DECL LDAT LCPDAT2987={VEL 2.00000,ACC 100.000,APO_DIST 500.000,APO_FAC 50.0000,AXIS_VEL 100.000,AXIS_ACC 100.000,ORI_TYP #VAR,CIRC_TYP #BASE,JERK_FAC 50.0000,GEAR_JERK 100.000,EXAX_IGN 0}
DECL E6POS XP2988={X 377.0,Y 306.0,Z -17.64,A -180,B 0,C 180,S 2,T 10,E1 0.0,E2 0.0,E3 0.0,E4 0.0,E5 0.0,E6 0.0}
DECL FDAT FP2988={TOOL_NO 1,BASE_NO 0,IPO_FRAME #BASE,POINT2[] " "}
DECL LDAT LCPDAT2988={VEL 2.00000,ACC 100.000,APO_DIST 500.000,APO_FAC 50.0000,AXIS_VEL 100.000,AXIS_ACC 100.000,ORI_TYP #VAR,CIRC_TYP #BASE,JERK_FAC 50.0000,GEAR_JERK 100.000,EXAX_IGN 0}
DECL E6POS XP2989={X 377.0,Y 306.0,Z -17.64,A -180,B 0,C 180,S 2,T 10,E1 0.0,E2 0.0,E3 0.0,E4 0.0,E5 0.0,E6 0.0}
DECL FDAT FP2989={TOOL_NO 1,BASE_NO 0,IPO_FRAME #BASE,POINT2[] " "}
DECL LDAT LCPDAT2989={VEL 2.00000,ACC 100.000,APO_DIST 500.000,APO_FAC 50.0000,AXIS_VEL 100.000,AXIS_ACC 100.000,ORI_TYP #VAR,CIRC_TYP #BASE,JERK_FAC 50.0000,GEAR_JERK 100.000,EXAX_IGN 0}
DECL E6POS XP2990={X 379.0,Y 306.0,Z -17.64,A -180,B 0,C 180,S 2,T 10,E1 0.0,E2 0.0,E3 0.0,E4 0.0,E5 0.0,E6 0.0}
DECL FDAT FP2990={TOOL_NO 1,BASE_NO 0,IPO_FRAME #BASE,POINT2[] " "}
DECL LDAT LCPDAT2990={VEL 2.00000,ACC 100.000,APO_DIST 500.000,APO_FAC 50.0000,AXIS_VEL 100.000,AXIS_ACC 100.000,ORI_TYP #VAR,CIRC_TYP #BASE,JERK_FAC 50.0000,GEAR_JERK 100.000,EXAX_IGN 0}
DECL E6POS XP2991={X 379.0,Y 306.0,Z -17.64,A -180,B 0,C 180,S 2,T 10,E1 0.0,E2 0.0,E3 0.0,E4 0.0,E5 0.0,E6 0.0}
DECL FDAT FP2991={TOOL_NO 1,BASE_NO 0,IPO_FRAME #BASE,POINT2[] " "}
DECL LDAT LCPDAT2991={VEL 2.00000,ACC 100.000,APO_DIST 500.000,APO_FAC 50.0000,AXIS_VEL 100.000,AXIS_ACC 100.000,ORI_TYP #VAR,CIRC_TYP #BASE,JERK_FAC 50.0000,GEAR_JERK 100.000,EXAX_IGN 0}
DECL E6POS XP2992={X 380.0,Y 304.0,Z -17.64,A -180,B 0,C 180,S 2,T 10,E1 0.0,E2 0.0,E3 0.0,E4 0.0,E5 0.0,E6 0.0}
DECL FDAT FP2992={TOOL_NO 1,BASE_NO 0,IPO_FRAME #BASE,POINT2[] " "}
DECL LDAT LCPDAT2992={VEL 2.00000,ACC 100.000,APO_DIST 500.000,APO_FAC 50.0000,AXIS_VEL 100.000,AXIS_ACC 100.000,ORI_TYP #VAR,CIRC_TYP #BASE,JERK_FAC 50.0000,GEAR_JERK 100.000,EXAX_IGN 0}
DECL E6POS XP2993={X 380.0,Y 304.0,Z -17.64,A -180,B 0,C 180,S 2,T 10,E1 0.0,E2 0.0,E3 0.0,E4 0.0,E5 0.0,E6 0.0}
DECL FDAT FP2993={TOOL_NO 1,BASE_NO 0,IPO_FRAME #BASE,POINT2[] " "}
DECL LDAT LCPDAT2993={VEL 2.00000,ACC 100.000,APO_DIST 500.000,APO_FAC 50.0000,AXIS_VEL 100.000,AXIS_ACC 100.000,ORI_TYP #VAR,CIRC_TYP #BASE,JERK_FAC 50.0000,GEAR_JERK 100.000,EXAX_IGN 0}
DECL E6POS XP2994={X 381.0,Y 313.0,Z -17.64,A -180,B 0,C 180,S 2,T 10,E1 0.0,E2 0.0,E3 0.0,E4 0.0,E5 0.0,E6 0.0}
DECL FDAT FP2994={TOOL_NO 1,BASE_NO 0,IPO_FRAME #BASE,POINT2[] " "}
DECL LDAT LCPDAT2994={VEL 2.00000,ACC 100.000,APO_DIST 500.000,APO_FAC 50.0000,AXIS_VEL 100.000,AXIS_ACC 100.000,ORI_TYP #VAR,CIRC_TYP #BASE,JERK_FAC 50.0000,GEAR_JERK 100.000,EXAX_IGN 0}
DECL E6POS XP2995={X 381.0,Y 313.0,Z -17.64,A -180,B 0,C 180,S 2,T 10,E1 0.0,E2 0.0,E3 0.0,E4 0.0,E5 0.0,E6 0.0}
DECL FDAT FP2995={TOOL_NO 1,BASE_NO 0,IPO_FRAME #BASE,POINT2[] " "}
DECL LDAT LCPDAT2995={VEL 2.00000,ACC 100.000,APO_DIST 500.000,APO_FAC 50.0000,AXIS_VEL 100.000,AXIS_ACC 100.000,ORI_TYP #VAR,CIRC_TYP #BASE,JERK_FAC 50.0000,GEAR_JERK 100.000,EXAX_IGN 0}
DECL E6POS XP2996={X 379.0,Y 315.0,Z -17.64,A -180,B 0,C 180,S 2,T 10,E1 0.0,E2 0.0,E3 0.0,E4 0.0,E5 0.0,E6 0.0}
DECL FDAT FP2996={TOOL_NO 1,BASE_NO 0,IPO_FRAME #BASE,POINT2[] " "}
DECL LDAT LCPDAT2996={VEL 2.00000,ACC 100.000,APO_DIST 500.000,APO_FAC 50.0000,AXIS_VEL 100.000,AXIS_ACC 100.000,ORI_TYP #VAR,CIRC_TYP #BASE,JERK_FAC 50.0000,GEAR_JERK 100.000,EXAX_IGN 0}
DECL E6POS XP2997={X 379.0,Y 315.0,Z -17.64,A -180,B 0,C 180,S 2,T 10,E1 0.0,E2 0.0,E3 0.0,E4 0.0,E5 0.0,E6 0.0}
DECL FDAT FP2997={TOOL_NO 1,BASE_NO 0,IPO_FRAME #BASE,POINT2[] " "}
DECL LDAT LCPDAT2997={VEL 2.00000,ACC 100.000,APO_DIST 500.000,APO_FAC 50.0000,AXIS_VEL 100.000,AXIS_ACC 100.000,ORI_TYP #VAR,CIRC_TYP #BASE,JERK_FAC 50.0000,GEAR_JERK 100.000,EXAX_IGN 0}
DECL E6POS XP2998={X 375.0,Y 315.0,Z -17.64,A -180,B 0,C 180,S 2,T 10,E1 0.0,E2 0.0,E3 0.0,E4 0.0,E5 0.0,E6 0.0}
DECL FDAT FP2998={TOOL_NO 1,BASE_NO 0,IPO_FRAME #BASE,POINT2[] " "}
DECL LDAT LCPDAT2998={VEL 2.00000,ACC 100.000,APO_DIST 500.000,APO_FAC 50.0000,AXIS_VEL 100.000,AXIS_ACC 100.000,ORI_TYP #VAR,CIRC_TYP #BASE,JERK_FAC 50.0000,GEAR_JERK 100.000,EXAX_IGN 0}
DECL E6POS XP2999={X 375.0,Y 315.0,Z -17.64,A -180,B 0,C 180,S 2,T 10,E1 0.0,E2 0.0,E3 0.0,E4 0.0,E5 0.0,E6 0.0}
DECL FDAT FP2999={TOOL_NO 1,BASE_NO 0,IPO_FRAME #BASE,POINT2[] " "}
DECL LDAT LCPDAT2999={VEL 2.00000,ACC 100.000,APO_DIST 500.000,APO_FAC 50.0000,AXIS_VEL 100.000,AXIS_ACC 100.000,ORI_TYP #VAR,CIRC_TYP #BASE,JERK_FAC 50.0000,GEAR_JERK 100.000,EXAX_IGN 0}
DECL E6POS XP3000={X 375.0,Y 317.0,Z -17.64,A -180,B 0,C 180,S 2,T 10,E1 0.0,E2 0.0,E3 0.0,E4 0.0,E5 0.0,E6 0.0}
DECL FDAT FP3000={TOOL_NO 1,BASE_NO 0,IPO_FRAME #BASE,POINT2[] " "}
DECL LDAT LCPDAT3000={VEL 2.00000,ACC 100.000,APO_DIST 500.000,APO_FAC 50.0000,AXIS_VEL 100.000,AXIS_ACC 100.000,ORI_TYP #VAR,CIRC_TYP #BASE,JERK_FAC 50.0000,GEAR_JERK 100.000,EXAX_IGN 0}
DECL E6POS XP3001={X 375.0,Y 317.0,Z -17.64,A -180,B 0,C 180,S 2,T 10,E1 0.0,E2 0.0,E3 0.0,E4 0.0,E5 0.0,E6 0.0}
DECL FDAT FP3001={TOOL_NO 1,BASE_NO 0,IPO_FRAME #BASE,POINT2[] " "}
DECL LDAT LCPDAT3001={VEL 2.00000,ACC 100.000,APO_DIST 500.000,APO_FAC 50.0000,AXIS_VEL 100.000,AXIS_ACC 100.000,ORI_TYP #VAR,CIRC_TYP #BASE,JERK_FAC 50.0000,GEAR_JERK 100.000,EXAX_IGN 0}
DECL E6POS XP3002={X 376.0,Y 320.0,Z -17.64,A -180,B 0,C 180,S 2,T 10,E1 0.0,E2 0.0,E3 0.0,E4 0.0,E5 0.0,E6 0.0}
DECL FDAT FP3002={TOOL_NO 1,BASE_NO 0,IPO_FRAME #BASE,POINT2[] " "}
DECL LDAT LCPDAT3002={VEL 2.00000,ACC 100.000,APO_DIST 500.000,APO_FAC 50.0000,AXIS_VEL 100.000,AXIS_ACC 100.000,ORI_TYP #VAR,CIRC_TYP #BASE,JERK_FAC 50.0000,GEAR_JERK 100.000,EXAX_IGN 0}
DECL E6POS XP3003={X 376.0,Y 320.0,Z -17.64,A -180,B 0,C 180,S 2,T 10,E1 0.0,E2 0.0,E3 0.0,E4 0.0,E5 0.0,E6 0.0}
DECL FDAT FP3003={TOOL_NO 1,BASE_NO 0,IPO_FRAME #BASE,POINT2[] " "}
DECL LDAT LCPDAT3003={VEL 2.00000,ACC 100.000,APO_DIST 500.000,APO_FAC 50.0000,AXIS_VEL 100.000,AXIS_ACC 100.000,ORI_TYP #VAR,CIRC_TYP #BASE,JERK_FAC 50.0000,GEAR_JERK 100.000,EXAX_IGN 0}
DECL E6POS XP3004={X 378.0,Y 322.0,Z -17.64,A -180,B 0,C 180,S 2,T 10,E1 0.0,E2 0.0,E3 0.0,E4 0.0,E5 0.0,E6 0.0}
DECL FDAT FP3004={TOOL_NO 1,BASE_NO 0,IPO_FRAME #BASE,POINT2[] " "}
DECL LDAT LCPDAT3004={VEL 2.00000,ACC 100.000,APO_DIST 500.000,APO_FAC 50.0000,AXIS_VEL 100.000,AXIS_ACC 100.000,ORI_TYP #VAR,CIRC_TYP #BASE,JERK_FAC 50.0000,GEAR_JERK 100.000,EXAX_IGN 0}
DECL E6POS XP3005={X 378.0,Y 322.0,Z -17.64,A -180,B 0,C 180,S 2,T 10,E1 0.0,E2 0.0,E3 0.0,E4 0.0,E5 0.0,E6 0.0}
DECL FDAT FP3005={TOOL_NO 1,BASE_NO 0,IPO_FRAME #BASE,POINT2[] " "}
DECL LDAT LCPDAT3005={VEL 2.00000,ACC 100.000,APO_DIST 500.000,APO_FAC 50.0000,AXIS_VEL 100.000,AXIS_ACC 100.000,ORI_TYP #VAR,CIRC_TYP #BASE,JERK_FAC 50.0000,GEAR_JERK 100.000,EXAX_IGN 0}
DECL E6POS XP3006={X 379.0,Y 326.0,Z -17.64,A -180,B 0,C 180,S 2,T 10,E1 0.0,E2 0.0,E3 0.0,E4 0.0,E5 0.0,E6 0.0}
DECL FDAT FP3006={TOOL_NO 1,BASE_NO 0,IPO_FRAME #BASE,POINT2[] " "}
DECL LDAT LCPDAT3006={VEL 2.00000,ACC 100.000,APO_DIST 500.000,APO_FAC 50.0000,AXIS_VEL 100.000,AXIS_ACC 100.000,ORI_TYP #VAR,CIRC_TYP #BASE,JERK_FAC 50.0000,GEAR_JERK 100.000,EXAX_IGN 0}
DECL E6POS XP3007={X 379.0,Y 326.0,Z -17.64,A -180,B 0,C 180,S 2,T 10,E1 0.0,E2 0.0,E3 0.0,E4 0.0,E5 0.0,E6 0.0}
DECL FDAT FP3007={TOOL_NO 1,BASE_NO 0,IPO_FRAME #BASE,POINT2[] " "}
DECL LDAT LCPDAT3007={VEL 2.00000,ACC 100.000,APO_DIST 500.000,APO_FAC 50.0000,AXIS_VEL 100.000,AXIS_ACC 100.000,ORI_TYP #VAR,CIRC_TYP #BASE,JERK_FAC 50.0000,GEAR_JERK 100.000,EXAX_IGN 0}
DECL E6POS XP3008={X 378.0,Y 330.0,Z -17.64,A -180,B 0,C 180,S 2,T 10,E1 0.0,E2 0.0,E3 0.0,E4 0.0,E5 0.0,E6 0.0}
DECL FDAT FP3008={TOOL_NO 1,BASE_NO 0,IPO_FRAME #BASE,POINT2[] " "}
DECL LDAT LCPDAT3008={VEL 2.00000,ACC 100.000,APO_DIST 500.000,APO_FAC 50.0000,AXIS_VEL 100.000,AXIS_ACC 100.000,ORI_TYP #VAR,CIRC_TYP #BASE,JERK_FAC 50.0000,GEAR_JERK 100.000,EXAX_IGN 0}
DECL E6POS XP3009={X 378.0,Y 330.0,Z -17.64,A -180,B 0,C 180,S 2,T 10,E1 0.0,E2 0.0,E3 0.0,E4 0.0,E5 0.0,E6 0.0}
DECL FDAT FP3009={TOOL_NO 1,BASE_NO 0,IPO_FRAME #BASE,POINT2[] " "}
DECL LDAT LCPDAT3009={VEL 2.00000,ACC 100.000,APO_DIST 500.000,APO_FAC 50.0000,AXIS_VEL 100.000,AXIS_ACC 100.000,ORI_TYP #VAR,CIRC_TYP #BASE,JERK_FAC 50.0000,GEAR_JERK 100.000,EXAX_IGN 0}
DECL E6POS XP3010={X 376.0,Y 329.0,Z -17.64,A -180,B 0,C 180,S 2,T 10,E1 0.0,E2 0.0,E3 0.0,E4 0.0,E5 0.0,E6 0.0}
DECL FDAT FP3010={TOOL_NO 1,BASE_NO 0,IPO_FRAME #BASE,POINT2[] " "}
DECL LDAT LCPDAT3010={VEL 2.00000,ACC 100.000,APO_DIST 500.000,APO_FAC 50.0000,AXIS_VEL 100.000,AXIS_ACC 100.000,ORI_TYP #VAR,CIRC_TYP #BASE,JERK_FAC 50.0000,GEAR_JERK 100.000,EXAX_IGN 0}
DECL E6POS XP3011={X 376.0,Y 329.0,Z -17.64,A -180,B 0,C 180,S 2,T 10,E1 0.0,E2 0.0,E3 0.0,E4 0.0,E5 0.0,E6 0.0}
DECL FDAT FP3011={TOOL_NO 1,BASE_NO 0,IPO_FRAME #BASE,POINT2[] " "}
DECL LDAT LCPDAT3011={VEL 2.00000,ACC 100.000,APO_DIST 500.000,APO_FAC 50.0000,AXIS_VEL 100.000,AXIS_ACC 100.000,ORI_TYP #VAR,CIRC_TYP #BASE,JERK_FAC 50.0000,GEAR_JERK 100.000,EXAX_IGN 0}
DECL E6POS XP3012={X 376.0,Y 334.0,Z -17.64,A -180,B 0,C 180,S 2,T 10,E1 0.0,E2 0.0,E3 0.0,E4 0.0,E5 0.0,E6 0.0}
DECL FDAT FP3012={TOOL_NO 1,BASE_NO 0,IPO_FRAME #BASE,POINT2[] " "}
DECL LDAT LCPDAT3012={VEL 2.00000,ACC 100.000,APO_DIST 500.000,APO_FAC 50.0000,AXIS_VEL 100.000,AXIS_ACC 100.000,ORI_TYP #VAR,CIRC_TYP #BASE,JERK_FAC 50.0000,GEAR_JERK 100.000,EXAX_IGN 0}
DECL E6POS XP3013={X 376.0,Y 334.0,Z -17.64,A -180,B 0,C 180,S 2,T 10,E1 0.0,E2 0.0,E3 0.0,E4 0.0,E5 0.0,E6 0.0}
DECL FDAT FP3013={TOOL_NO 1,BASE_NO 0,IPO_FRAME #BASE,POINT2[] " "}
DECL LDAT LCPDAT3013={VEL 2.00000,ACC 100.000,APO_DIST 500.000,APO_FAC 50.0000,AXIS_VEL 100.000,AXIS_ACC 100.000,ORI_TYP #VAR,CIRC_TYP #BASE,JERK_FAC 50.0000,GEAR_JERK 100.000,EXAX_IGN 0}
DECL E6POS XP3014={X 378.0,Y 333.0,Z -17.64,A -180,B 0,C 180,S 2,T 10,E1 0.0,E2 0.0,E3 0.0,E4 0.0,E5 0.0,E6 0.0}
DECL FDAT FP3014={TOOL_NO 1,BASE_NO 0,IPO_FRAME #BASE,POINT2[] " "}
DECL LDAT LCPDAT3014={VEL 2.00000,ACC 100.000,APO_DIST 500.000,APO_FAC 50.0000,AXIS_VEL 100.000,AXIS_ACC 100.000,ORI_TYP #VAR,CIRC_TYP #BASE,JERK_FAC 50.0000,GEAR_JERK 100.000,EXAX_IGN 0}
DECL E6POS XP3015={X 378.0,Y 333.0,Z -17.64,A -180,B 0,C 180,S 2,T 10,E1 0.0,E2 0.0,E3 0.0,E4 0.0,E5 0.0,E6 0.0}
DECL FDAT FP3015={TOOL_NO 1,BASE_NO 0,IPO_FRAME #BASE,POINT2[] " "}
DECL LDAT LCPDAT3015={VEL 2.00000,ACC 100.000,APO_DIST 500.000,APO_FAC 50.0000,AXIS_VEL 100.000,AXIS_ACC 100.000,ORI_TYP #VAR,CIRC_TYP #BASE,JERK_FAC 50.0000,GEAR_JERK 100.000,EXAX_IGN 0}
DECL E6POS XP3016={X 378.0,Y 337.0,Z -17.64,A -180,B 0,C 180,S 2,T 10,E1 0.0,E2 0.0,E3 0.0,E4 0.0,E5 0.0,E6 0.0}
DECL FDAT FP3016={TOOL_NO 1,BASE_NO 0,IPO_FRAME #BASE,POINT2[] " "}
DECL LDAT LCPDAT3016={VEL 2.00000,ACC 100.000,APO_DIST 500.000,APO_FAC 50.0000,AXIS_VEL 100.000,AXIS_ACC 100.000,ORI_TYP #VAR,CIRC_TYP #BASE,JERK_FAC 50.0000,GEAR_JERK 100.000,EXAX_IGN 0}
DECL E6POS XP3017={X 378.0,Y 337.0,Z -17.64,A -180,B 0,C 180,S 2,T 10,E1 0.0,E2 0.0,E3 0.0,E4 0.0,E5 0.0,E6 0.0}
DECL FDAT FP3017={TOOL_NO 1,BASE_NO 0,IPO_FRAME #BASE,POINT2[] " "}
DECL LDAT LCPDAT3017={VEL 2.00000,ACC 100.000,APO_DIST 500.000,APO_FAC 50.0000,AXIS_VEL 100.000,AXIS_ACC 100.000,ORI_TYP #VAR,CIRC_TYP #BASE,JERK_FAC 50.0000,GEAR_JERK 100.000,EXAX_IGN 0}
DECL E6POS XP3018={X 377.0,Y 336.0,Z -17.64,A -180,B 0,C 180,S 2,T 10,E1 0.0,E2 0.0,E3 0.0,E4 0.0,E5 0.0,E6 0.0}
DECL FDAT FP3018={TOOL_NO 1,BASE_NO 0,IPO_FRAME #BASE,POINT2[] " "}
DECL LDAT LCPDAT3018={VEL 2.00000,ACC 100.000,APO_DIST 500.000,APO_FAC 50.0000,AXIS_VEL 100.000,AXIS_ACC 100.000,ORI_TYP #VAR,CIRC_TYP #BASE,JERK_FAC 50.0000,GEAR_JERK 100.000,EXAX_IGN 0}
DECL E6POS XP3019={X 377.0,Y 336.0,Z -17.64,A -180,B 0,C 180,S 2,T 10,E1 0.0,E2 0.0,E3 0.0,E4 0.0,E5 0.0,E6 0.0}
DECL FDAT FP3019={TOOL_NO 1,BASE_NO 0,IPO_FRAME #BASE,POINT2[] " "}
DECL LDAT LCPDAT3019={VEL 2.00000,ACC 100.000,APO_DIST 500.000,APO_FAC 50.0000,AXIS_VEL 100.000,AXIS_ACC 100.000,ORI_TYP #VAR,CIRC_TYP #BASE,JERK_FAC 50.0000,GEAR_JERK 100.000,EXAX_IGN 0}
DECL E6POS XP3020={X 376.0,Y 339.0,Z -17.64,A -180,B 0,C 180,S 2,T 10,E1 0.0,E2 0.0,E3 0.0,E4 0.0,E5 0.0,E6 0.0}
DECL FDAT FP3020={TOOL_NO 1,BASE_NO 0,IPO_FRAME #BASE,POINT2[] " "}
DECL LDAT LCPDAT3020={VEL 2.00000,ACC 100.000,APO_DIST 500.000,APO_FAC 50.0000,AXIS_VEL 100.000,AXIS_ACC 100.000,ORI_TYP #VAR,CIRC_TYP #BASE,JERK_FAC 50.0000,GEAR_JERK 100.000,EXAX_IGN 0}
DECL E6POS XP3021={X 376.0,Y 339.0,Z -17.64,A -180,B 0,C 180,S 2,T 10,E1 0.0,E2 0.0,E3 0.0,E4 0.0,E5 0.0,E6 0.0}
DECL FDAT FP3021={TOOL_NO 1,BASE_NO 0,IPO_FRAME #BASE,POINT2[] " "}
DECL LDAT LCPDAT3021={VEL 2.00000,ACC 100.000,APO_DIST 500.000,APO_FAC 50.0000,AXIS_VEL 100.000,AXIS_ACC 100.000,ORI_TYP #VAR,CIRC_TYP #BASE,JERK_FAC 50.0000,GEAR_JERK 100.000,EXAX_IGN 0}
DECL E6POS XP3022={X 374.0,Y 341.0,Z -17.64,A -180,B 0,C 180,S 2,T 10,E1 0.0,E2 0.0,E3 0.0,E4 0.0,E5 0.0,E6 0.0}
DECL FDAT FP3022={TOOL_NO 1,BASE_NO 0,IPO_FRAME #BASE,POINT2[] " "}
DECL LDAT LCPDAT3022={VEL 2.00000,ACC 100.000,APO_DIST 500.000,APO_FAC 50.0000,AXIS_VEL 100.000,AXIS_ACC 100.000,ORI_TYP #VAR,CIRC_TYP #BASE,JERK_FAC 50.0000,GEAR_JERK 100.000,EXAX_IGN 0}
DECL E6POS XP3023={X 374.0,Y 341.0,Z -17.64,A -180,B 0,C 180,S 2,T 10,E1 0.0,E2 0.0,E3 0.0,E4 0.0,E5 0.0,E6 0.0}
DECL FDAT FP3023={TOOL_NO 1,BASE_NO 0,IPO_FRAME #BASE,POINT2[] " "}
DECL LDAT LCPDAT3023={VEL 2.00000,ACC 100.000,APO_DIST 500.000,APO_FAC 50.0000,AXIS_VEL 100.000,AXIS_ACC 100.000,ORI_TYP #VAR,CIRC_TYP #BASE,JERK_FAC 50.0000,GEAR_JERK 100.000,EXAX_IGN 0}
DECL E6POS XP3024={X 372.0,Y 338.0,Z -17.64,A -180,B 0,C 180,S 2,T 10,E1 0.0,E2 0.0,E3 0.0,E4 0.0,E5 0.0,E6 0.0}
DECL FDAT FP3024={TOOL_NO 1,BASE_NO 0,IPO_FRAME #BASE,POINT2[] " "}
DECL LDAT LCPDAT3024={VEL 2.00000,ACC 100.000,APO_DIST 500.000,APO_FAC 50.0000,AXIS_VEL 100.000,AXIS_ACC 100.000,ORI_TYP #VAR,CIRC_TYP #BASE,JERK_FAC 50.0000,GEAR_JERK 100.000,EXAX_IGN 0}
DECL E6POS XP3025={X 372.0,Y 338.0,Z -17.64,A -180,B 0,C 180,S 2,T 10,E1 0.0,E2 0.0,E3 0.0,E4 0.0,E5 0.0,E6 0.0}
DECL FDAT FP3025={TOOL_NO 1,BASE_NO 0,IPO_FRAME #BASE,POINT2[] " "}
DECL LDAT LCPDAT3025={VEL 2.00000,ACC 100.000,APO_DIST 500.000,APO_FAC 50.0000,AXIS_VEL 100.000,AXIS_ACC 100.000,ORI_TYP #VAR,CIRC_TYP #BASE,JERK_FAC 50.0000,GEAR_JERK 100.000,EXAX_IGN 0}
DECL E6POS XP3026={X 374.0,Y 337.0,Z -17.64,A -180,B 0,C 180,S 2,T 10,E1 0.0,E2 0.0,E3 0.0,E4 0.0,E5 0.0,E6 0.0}
DECL FDAT FP3026={TOOL_NO 1,BASE_NO 0,IPO_FRAME #BASE,POINT2[] " "}
DECL LDAT LCPDAT3026={VEL 2.00000,ACC 100.000,APO_DIST 500.000,APO_FAC 50.0000,AXIS_VEL 100.000,AXIS_ACC 100.000,ORI_TYP #VAR,CIRC_TYP #BASE,JERK_FAC 50.0000,GEAR_JERK 100.000,EXAX_IGN 0}
DECL E6POS XP3027={X 374.0,Y 337.0,Z -17.64,A -180,B 0,C 180,S 2,T 10,E1 0.0,E2 0.0,E3 0.0,E4 0.0,E5 0.0,E6 0.0}
DECL FDAT FP3027={TOOL_NO 1,BASE_NO 0,IPO_FRAME #BASE,POINT2[] " "}
DECL LDAT LCPDAT3027={VEL 2.00000,ACC 100.000,APO_DIST 500.000,APO_FAC 50.0000,AXIS_VEL 100.000,AXIS_ACC 100.000,ORI_TYP #VAR,CIRC_TYP #BASE,JERK_FAC 50.0000,GEAR_JERK 100.000,EXAX_IGN 0}
DECL E6POS XP3028={X 372.0,Y 338.0,Z -17.64,A -180,B 0,C 180,S 2,T 10,E1 0.0,E2 0.0,E3 0.0,E4 0.0,E5 0.0,E6 0.0}
DECL FDAT FP3028={TOOL_NO 1,BASE_NO 0,IPO_FRAME #BASE,POINT2[] " "}
DECL LDAT LCPDAT3028={VEL 2.00000,ACC 100.000,APO_DIST 500.000,APO_FAC 50.0000,AXIS_VEL 100.000,AXIS_ACC 100.000,ORI_TYP #VAR,CIRC_TYP #BASE,JERK_FAC 50.0000,GEAR_JERK 100.000,EXAX_IGN 0}
DECL E6POS XP3029={X 372.0,Y 338.0,Z -17.64,A -180,B 0,C 180,S 2,T 10,E1 0.0,E2 0.0,E3 0.0,E4 0.0,E5 0.0,E6 0.0}
DECL FDAT FP3029={TOOL_NO 1,BASE_NO 0,IPO_FRAME #BASE,POINT2[] " "}
DECL LDAT LCPDAT3029={VEL 2.00000,ACC 100.000,APO_DIST 500.000,APO_FAC 50.0000,AXIS_VEL 100.000,AXIS_ACC 100.000,ORI_TYP #VAR,CIRC_TYP #BASE,JERK_FAC 50.0000,GEAR_JERK 100.000,EXAX_IGN 0}
DECL E6POS XP3030={X 373.0,Y 341.0,Z -17.64,A -180,B 0,C 180,S 2,T 10,E1 0.0,E2 0.0,E3 0.0,E4 0.0,E5 0.0,E6 0.0}
DECL FDAT FP3030={TOOL_NO 1,BASE_NO 0,IPO_FRAME #BASE,POINT2[] " "}
DECL LDAT LCPDAT3030={VEL 2.00000,ACC 100.000,APO_DIST 500.000,APO_FAC 50.0000,AXIS_VEL 100.000,AXIS_ACC 100.000,ORI_TYP #VAR,CIRC_TYP #BASE,JERK_FAC 50.0000,GEAR_JERK 100.000,EXAX_IGN 0}
DECL E6POS XP3031={X 373.0,Y 341.0,Z -17.64,A -180,B 0,C 180,S 2,T 10,E1 0.0,E2 0.0,E3 0.0,E4 0.0,E5 0.0,E6 0.0}
DECL FDAT FP3031={TOOL_NO 1,BASE_NO 0,IPO_FRAME #BASE,POINT2[] " "}
DECL LDAT LCPDAT3031={VEL 2.00000,ACC 100.000,APO_DIST 500.000,APO_FAC 50.0000,AXIS_VEL 100.000,AXIS_ACC 100.000,ORI_TYP #VAR,CIRC_TYP #BASE,JERK_FAC 50.0000,GEAR_JERK 100.000,EXAX_IGN 0}
DECL E6POS XP3032={X 375.0,Y 342.0,Z -17.64,A -180,B 0,C 180,S 2,T 10,E1 0.0,E2 0.0,E3 0.0,E4 0.0,E5 0.0,E6 0.0}
DECL FDAT FP3032={TOOL_NO 1,BASE_NO 0,IPO_FRAME #BASE,POINT2[] " "}
DECL LDAT LCPDAT3032={VEL 2.00000,ACC 100.000,APO_DIST 500.000,APO_FAC 50.0000,AXIS_VEL 100.000,AXIS_ACC 100.000,ORI_TYP #VAR,CIRC_TYP #BASE,JERK_FAC 50.0000,GEAR_JERK 100.000,EXAX_IGN 0}
DECL E6POS XP3033={X 375.0,Y 342.0,Z -17.64,A -180,B 0,C 180,S 2,T 10,E1 0.0,E2 0.0,E3 0.0,E4 0.0,E5 0.0,E6 0.0}
DECL FDAT FP3033={TOOL_NO 1,BASE_NO 0,IPO_FRAME #BASE,POINT2[] " "}
DECL LDAT LCPDAT3033={VEL 2.00000,ACC 100.000,APO_DIST 500.000,APO_FAC 50.0000,AXIS_VEL 100.000,AXIS_ACC 100.000,ORI_TYP #VAR,CIRC_TYP #BASE,JERK_FAC 50.0000,GEAR_JERK 100.000,EXAX_IGN 0}
DECL E6POS XP3034={X 375.0,Y 344.0,Z -17.64,A -180,B 0,C 180,S 2,T 10,E1 0.0,E2 0.0,E3 0.0,E4 0.0,E5 0.0,E6 0.0}
DECL FDAT FP3034={TOOL_NO 1,BASE_NO 0,IPO_FRAME #BASE,POINT2[] " "}
DECL LDAT LCPDAT3034={VEL 2.00000,ACC 100.000,APO_DIST 500.000,APO_FAC 50.0000,AXIS_VEL 100.000,AXIS_ACC 100.000,ORI_TYP #VAR,CIRC_TYP #BASE,JERK_FAC 50.0000,GEAR_JERK 100.000,EXAX_IGN 0}
DECL E6POS XP3035={X 375.0,Y 344.0,Z -17.64,A -180,B 0,C 180,S 2,T 10,E1 0.0,E2 0.0,E3 0.0,E4 0.0,E5 0.0,E6 0.0}
DECL FDAT FP3035={TOOL_NO 1,BASE_NO 0,IPO_FRAME #BASE,POINT2[] " "}
DECL LDAT LCPDAT3035={VEL 2.00000,ACC 100.000,APO_DIST 500.000,APO_FAC 50.0000,AXIS_VEL 100.000,AXIS_ACC 100.000,ORI_TYP #VAR,CIRC_TYP #BASE,JERK_FAC 50.0000,GEAR_JERK 100.000,EXAX_IGN 0}
DECL E6POS XP3036={X 380.0,Y 350.0,Z -17.64,A -180,B 0,C 180,S 2,T 10,E1 0.0,E2 0.0,E3 0.0,E4 0.0,E5 0.0,E6 0.0}
DECL FDAT FP3036={TOOL_NO 1,BASE_NO 0,IPO_FRAME #BASE,POINT2[] " "}
DECL LDAT LCPDAT3036={VEL 2.00000,ACC 100.000,APO_DIST 500.000,APO_FAC 50.0000,AXIS_VEL 100.000,AXIS_ACC 100.000,ORI_TYP #VAR,CIRC_TYP #BASE,JERK_FAC 50.0000,GEAR_JERK 100.000,EXAX_IGN 0}
DECL E6POS XP3037={X 380.0,Y 350.0,Z -17.64,A -180,B 0,C 180,S 2,T 10,E1 0.0,E2 0.0,E3 0.0,E4 0.0,E5 0.0,E6 0.0}
DECL FDAT FP3037={TOOL_NO 1,BASE_NO 0,IPO_FRAME #BASE,POINT2[] " "}
DECL LDAT LCPDAT3037={VEL 2.00000,ACC 100.000,APO_DIST 500.000,APO_FAC 50.0000,AXIS_VEL 100.000,AXIS_ACC 100.000,ORI_TYP #VAR,CIRC_TYP #BASE,JERK_FAC 50.0000,GEAR_JERK 100.000,EXAX_IGN 0}
DECL E6POS XP3038={X 382.0,Y 353.0,Z -17.64,A -180,B 0,C 180,S 2,T 10,E1 0.0,E2 0.0,E3 0.0,E4 0.0,E5 0.0,E6 0.0}
DECL FDAT FP3038={TOOL_NO 1,BASE_NO 0,IPO_FRAME #BASE,POINT2[] " "}
DECL LDAT LCPDAT3038={VEL 2.00000,ACC 100.000,APO_DIST 500.000,APO_FAC 50.0000,AXIS_VEL 100.000,AXIS_ACC 100.000,ORI_TYP #VAR,CIRC_TYP #BASE,JERK_FAC 50.0000,GEAR_JERK 100.000,EXAX_IGN 0}
DECL E6POS XP3039={X 382.0,Y 353.0,Z -17.64,A -180,B 0,C 180,S 2,T 10,E1 0.0,E2 0.0,E3 0.0,E4 0.0,E5 0.0,E6 0.0}
DECL FDAT FP3039={TOOL_NO 1,BASE_NO 0,IPO_FRAME #BASE,POINT2[] " "}
DECL LDAT LCPDAT3039={VEL 2.00000,ACC 100.000,APO_DIST 500.000,APO_FAC 50.0000,AXIS_VEL 100.000,AXIS_ACC 100.000,ORI_TYP #VAR,CIRC_TYP #BASE,JERK_FAC 50.0000,GEAR_JERK 100.000,EXAX_IGN 0}
DECL E6POS XP3040={X 380.0,Y 351.0,Z -17.64,A -180,B 0,C 180,S 2,T 10,E1 0.0,E2 0.0,E3 0.0,E4 0.0,E5 0.0,E6 0.0}
DECL FDAT FP3040={TOOL_NO 1,BASE_NO 0,IPO_FRAME #BASE,POINT2[] " "}
DECL LDAT LCPDAT3040={VEL 2.00000,ACC 100.000,APO_DIST 500.000,APO_FAC 50.0000,AXIS_VEL 100.000,AXIS_ACC 100.000,ORI_TYP #VAR,CIRC_TYP #BASE,JERK_FAC 50.0000,GEAR_JERK 100.000,EXAX_IGN 0}
DECL E6POS XP3041={X 380.0,Y 351.0,Z -17.64,A -180,B 0,C 180,S 2,T 10,E1 0.0,E2 0.0,E3 0.0,E4 0.0,E5 0.0,E6 0.0}
DECL FDAT FP3041={TOOL_NO 1,BASE_NO 0,IPO_FRAME #BASE,POINT2[] " "}
DECL LDAT LCPDAT3041={VEL 2.00000,ACC 100.000,APO_DIST 500.000,APO_FAC 50.0000,AXIS_VEL 100.000,AXIS_ACC 100.000,ORI_TYP #VAR,CIRC_TYP #BASE,JERK_FAC 50.0000,GEAR_JERK 100.000,EXAX_IGN 0}
DECL E6POS XP3042={X 379.0,Y 349.0,Z -17.64,A -180,B 0,C 180,S 2,T 10,E1 0.0,E2 0.0,E3 0.0,E4 0.0,E5 0.0,E6 0.0}
DECL FDAT FP3042={TOOL_NO 1,BASE_NO 0,IPO_FRAME #BASE,POINT2[] " "}
DECL LDAT LCPDAT3042={VEL 2.00000,ACC 100.000,APO_DIST 500.000,APO_FAC 50.0000,AXIS_VEL 100.000,AXIS_ACC 100.000,ORI_TYP #VAR,CIRC_TYP #BASE,JERK_FAC 50.0000,GEAR_JERK 100.000,EXAX_IGN 0}
DECL E6POS XP3043={X 379.0,Y 349.0,Z -17.64,A -180,B 0,C 180,S 2,T 10,E1 0.0,E2 0.0,E3 0.0,E4 0.0,E5 0.0,E6 0.0}
DECL FDAT FP3043={TOOL_NO 1,BASE_NO 0,IPO_FRAME #BASE,POINT2[] " "}
DECL LDAT LCPDAT3043={VEL 2.00000,ACC 100.000,APO_DIST 500.000,APO_FAC 50.0000,AXIS_VEL 100.000,AXIS_ACC 100.000,ORI_TYP #VAR,CIRC_TYP #BASE,JERK_FAC 50.0000,GEAR_JERK 100.000,EXAX_IGN 0}
DECL E6POS XP3044={X 381.0,Y 347.0,Z -17.64,A -180,B 0,C 180,S 2,T 10,E1 0.0,E2 0.0,E3 0.0,E4 0.0,E5 0.0,E6 0.0}
DECL FDAT FP3044={TOOL_NO 1,BASE_NO 0,IPO_FRAME #BASE,POINT2[] " "}
DECL LDAT LCPDAT3044={VEL 2.00000,ACC 100.000,APO_DIST 500.000,APO_FAC 50.0000,AXIS_VEL 100.000,AXIS_ACC 100.000,ORI_TYP #VAR,CIRC_TYP #BASE,JERK_FAC 50.0000,GEAR_JERK 100.000,EXAX_IGN 0}
DECL E6POS XP3045={X 381.0,Y 347.0,Z -17.64,A -180,B 0,C 180,S 2,T 10,E1 0.0,E2 0.0,E3 0.0,E4 0.0,E5 0.0,E6 0.0}
DECL FDAT FP3045={TOOL_NO 1,BASE_NO 0,IPO_FRAME #BASE,POINT2[] " "}
DECL LDAT LCPDAT3045={VEL 2.00000,ACC 100.000,APO_DIST 500.000,APO_FAC 50.0000,AXIS_VEL 100.000,AXIS_ACC 100.000,ORI_TYP #VAR,CIRC_TYP #BASE,JERK_FAC 50.0000,GEAR_JERK 100.000,EXAX_IGN 0}
DECL E6POS XP3046={X 384.0,Y 351.0,Z -17.64,A -180,B 0,C 180,S 2,T 10,E1 0.0,E2 0.0,E3 0.0,E4 0.0,E5 0.0,E6 0.0}
DECL FDAT FP3046={TOOL_NO 1,BASE_NO 0,IPO_FRAME #BASE,POINT2[] " "}
DECL LDAT LCPDAT3046={VEL 2.00000,ACC 100.000,APO_DIST 500.000,APO_FAC 50.0000,AXIS_VEL 100.000,AXIS_ACC 100.000,ORI_TYP #VAR,CIRC_TYP #BASE,JERK_FAC 50.0000,GEAR_JERK 100.000,EXAX_IGN 0}
DECL E6POS XP3047={X 384.0,Y 351.0,Z -17.64,A -180,B 0,C 180,S 2,T 10,E1 0.0,E2 0.0,E3 0.0,E4 0.0,E5 0.0,E6 0.0}
DECL FDAT FP3047={TOOL_NO 1,BASE_NO 0,IPO_FRAME #BASE,POINT2[] " "}
DECL LDAT LCPDAT3047={VEL 2.00000,ACC 100.000,APO_DIST 500.000,APO_FAC 50.0000,AXIS_VEL 100.000,AXIS_ACC 100.000,ORI_TYP #VAR,CIRC_TYP #BASE,JERK_FAC 50.0000,GEAR_JERK 100.000,EXAX_IGN 0}
DECL E6POS XP3048={X 385.0,Y 354.0,Z -17.64,A -180,B 0,C 180,S 2,T 10,E1 0.0,E2 0.0,E3 0.0,E4 0.0,E5 0.0,E6 0.0}
DECL FDAT FP3048={TOOL_NO 1,BASE_NO 0,IPO_FRAME #BASE,POINT2[] " "}
DECL LDAT LCPDAT3048={VEL 2.00000,ACC 100.000,APO_DIST 500.000,APO_FAC 50.0000,AXIS_VEL 100.000,AXIS_ACC 100.000,ORI_TYP #VAR,CIRC_TYP #BASE,JERK_FAC 50.0000,GEAR_JERK 100.000,EXAX_IGN 0}
DECL E6POS XP3049={X 385.0,Y 354.0,Z -17.64,A -180,B 0,C 180,S 2,T 10,E1 0.0,E2 0.0,E3 0.0,E4 0.0,E5 0.0,E6 0.0}
DECL FDAT FP3049={TOOL_NO 1,BASE_NO 0,IPO_FRAME #BASE,POINT2[] " "}
DECL LDAT LCPDAT3049={VEL 2.00000,ACC 100.000,APO_DIST 500.000,APO_FAC 50.0000,AXIS_VEL 100.000,AXIS_ACC 100.000,ORI_TYP #VAR,CIRC_TYP #BASE,JERK_FAC 50.0000,GEAR_JERK 100.000,EXAX_IGN 0}
DECL E6POS XP3050={X 385.0,Y 359.0,Z -17.64,A -180,B 0,C 180,S 2,T 10,E1 0.0,E2 0.0,E3 0.0,E4 0.0,E5 0.0,E6 0.0}
DECL FDAT FP3050={TOOL_NO 1,BASE_NO 0,IPO_FRAME #BASE,POINT2[] " "}
DECL LDAT LCPDAT3050={VEL 2.00000,ACC 100.000,APO_DIST 500.000,APO_FAC 50.0000,AXIS_VEL 100.000,AXIS_ACC 100.000,ORI_TYP #VAR,CIRC_TYP #BASE,JERK_FAC 50.0000,GEAR_JERK 100.000,EXAX_IGN 0}
DECL E6POS XP3051={X 385.0,Y 359.0,Z -17.64,A -180,B 0,C 180,S 2,T 10,E1 0.0,E2 0.0,E3 0.0,E4 0.0,E5 0.0,E6 0.0}
DECL FDAT FP3051={TOOL_NO 1,BASE_NO 0,IPO_FRAME #BASE,POINT2[] " "}
DECL LDAT LCPDAT3051={VEL 2.00000,ACC 100.000,APO_DIST 500.000,APO_FAC 50.0000,AXIS_VEL 100.000,AXIS_ACC 100.000,ORI_TYP #VAR,CIRC_TYP #BASE,JERK_FAC 50.0000,GEAR_JERK 100.000,EXAX_IGN 0}
DECL E6POS XP3052={X 380.0,Y 364.0,Z -17.64,A -180,B 0,C 180,S 2,T 10,E1 0.0,E2 0.0,E3 0.0,E4 0.0,E5 0.0,E6 0.0}
DECL FDAT FP3052={TOOL_NO 1,BASE_NO 0,IPO_FRAME #BASE,POINT2[] " "}
DECL LDAT LCPDAT3052={VEL 2.00000,ACC 100.000,APO_DIST 500.000,APO_FAC 50.0000,AXIS_VEL 100.000,AXIS_ACC 100.000,ORI_TYP #VAR,CIRC_TYP #BASE,JERK_FAC 50.0000,GEAR_JERK 100.000,EXAX_IGN 0}
DECL E6POS XP3053={X 380.0,Y 364.0,Z -17.64,A -180,B 0,C 180,S 2,T 10,E1 0.0,E2 0.0,E3 0.0,E4 0.0,E5 0.0,E6 0.0}
DECL FDAT FP3053={TOOL_NO 1,BASE_NO 0,IPO_FRAME #BASE,POINT2[] " "}
DECL LDAT LCPDAT3053={VEL 2.00000,ACC 100.000,APO_DIST 500.000,APO_FAC 50.0000,AXIS_VEL 100.000,AXIS_ACC 100.000,ORI_TYP #VAR,CIRC_TYP #BASE,JERK_FAC 50.0000,GEAR_JERK 100.000,EXAX_IGN 0}
DECL E6POS XP3054={X 369.0,Y 371.0,Z -17.64,A -180,B 0,C 180,S 2,T 10,E1 0.0,E2 0.0,E3 0.0,E4 0.0,E5 0.0,E6 0.0}
DECL FDAT FP3054={TOOL_NO 1,BASE_NO 0,IPO_FRAME #BASE,POINT2[] " "}
DECL LDAT LCPDAT3054={VEL 2.00000,ACC 100.000,APO_DIST 500.000,APO_FAC 50.0000,AXIS_VEL 100.000,AXIS_ACC 100.000,ORI_TYP #VAR,CIRC_TYP #BASE,JERK_FAC 50.0000,GEAR_JERK 100.000,EXAX_IGN 0}
DECL E6POS XP3055={X 369.0,Y 371.0,Z -17.64,A -180,B 0,C 180,S 2,T 10,E1 0.0,E2 0.0,E3 0.0,E4 0.0,E5 0.0,E6 0.0}
DECL FDAT FP3055={TOOL_NO 1,BASE_NO 0,IPO_FRAME #BASE,POINT2[] " "}
DECL LDAT LCPDAT3055={VEL 2.00000,ACC 100.000,APO_DIST 500.000,APO_FAC 50.0000,AXIS_VEL 100.000,AXIS_ACC 100.000,ORI_TYP #VAR,CIRC_TYP #BASE,JERK_FAC 50.0000,GEAR_JERK 100.000,EXAX_IGN 0}
DECL E6POS XP3056={X 366.0,Y 372.0,Z -17.64,A -180,B 0,C 180,S 2,T 10,E1 0.0,E2 0.0,E3 0.0,E4 0.0,E5 0.0,E6 0.0}
DECL FDAT FP3056={TOOL_NO 1,BASE_NO 0,IPO_FRAME #BASE,POINT2[] " "}
DECL LDAT LCPDAT3056={VEL 2.00000,ACC 100.000,APO_DIST 500.000,APO_FAC 50.0000,AXIS_VEL 100.000,AXIS_ACC 100.000,ORI_TYP #VAR,CIRC_TYP #BASE,JERK_FAC 50.0000,GEAR_JERK 100.000,EXAX_IGN 0}
DECL E6POS XP3057={X 366.0,Y 372.0,Z -17.64,A -180,B 0,C 180,S 2,T 10,E1 0.0,E2 0.0,E3 0.0,E4 0.0,E5 0.0,E6 0.0}
DECL FDAT FP3057={TOOL_NO 1,BASE_NO 0,IPO_FRAME #BASE,POINT2[] " "}
DECL LDAT LCPDAT3057={VEL 2.00000,ACC 100.000,APO_DIST 500.000,APO_FAC 50.0000,AXIS_VEL 100.000,AXIS_ACC 100.000,ORI_TYP #VAR,CIRC_TYP #BASE,JERK_FAC 50.0000,GEAR_JERK 100.000,EXAX_IGN 0}
DECL E6POS XP3058={X 364.0,Y 370.0,Z -17.64,A -180,B 0,C 180,S 2,T 10,E1 0.0,E2 0.0,E3 0.0,E4 0.0,E5 0.0,E6 0.0}
DECL FDAT FP3058={TOOL_NO 1,BASE_NO 0,IPO_FRAME #BASE,POINT2[] " "}
DECL LDAT LCPDAT3058={VEL 2.00000,ACC 100.000,APO_DIST 500.000,APO_FAC 50.0000,AXIS_VEL 100.000,AXIS_ACC 100.000,ORI_TYP #VAR,CIRC_TYP #BASE,JERK_FAC 50.0000,GEAR_JERK 100.000,EXAX_IGN 0}
DECL E6POS XP3059={X 364.0,Y 370.0,Z -17.64,A -180,B 0,C 180,S 2,T 10,E1 0.0,E2 0.0,E3 0.0,E4 0.0,E5 0.0,E6 0.0}
DECL FDAT FP3059={TOOL_NO 1,BASE_NO 0,IPO_FRAME #BASE,POINT2[] " "}
DECL LDAT LCPDAT3059={VEL 2.00000,ACC 100.000,APO_DIST 500.000,APO_FAC 50.0000,AXIS_VEL 100.000,AXIS_ACC 100.000,ORI_TYP #VAR,CIRC_TYP #BASE,JERK_FAC 50.0000,GEAR_JERK 100.000,EXAX_IGN 0}
DECL E6POS XP3060={X 367.0,Y 369.0,Z -17.64,A -180,B 0,C 180,S 2,T 10,E1 0.0,E2 0.0,E3 0.0,E4 0.0,E5 0.0,E6 0.0}
DECL FDAT FP3060={TOOL_NO 1,BASE_NO 0,IPO_FRAME #BASE,POINT2[] " "}
DECL LDAT LCPDAT3060={VEL 2.00000,ACC 100.000,APO_DIST 500.000,APO_FAC 50.0000,AXIS_VEL 100.000,AXIS_ACC 100.000,ORI_TYP #VAR,CIRC_TYP #BASE,JERK_FAC 50.0000,GEAR_JERK 100.000,EXAX_IGN 0}
DECL E6POS XP3061={X 367.0,Y 369.0,Z -17.64,A -180,B 0,C 180,S 2,T 10,E1 0.0,E2 0.0,E3 0.0,E4 0.0,E5 0.0,E6 0.0}
DECL FDAT FP3061={TOOL_NO 1,BASE_NO 0,IPO_FRAME #BASE,POINT2[] " "}
DECL LDAT LCPDAT3061={VEL 2.00000,ACC 100.000,APO_DIST 500.000,APO_FAC 50.0000,AXIS_VEL 100.000,AXIS_ACC 100.000,ORI_TYP #VAR,CIRC_TYP #BASE,JERK_FAC 50.0000,GEAR_JERK 100.000,EXAX_IGN 0}
DECL E6POS XP3062={X 365.0,Y 368.0,Z -17.64,A -180,B 0,C 180,S 2,T 10,E1 0.0,E2 0.0,E3 0.0,E4 0.0,E5 0.0,E6 0.0}
DECL FDAT FP3062={TOOL_NO 1,BASE_NO 0,IPO_FRAME #BASE,POINT2[] " "}
DECL LDAT LCPDAT3062={VEL 2.00000,ACC 100.000,APO_DIST 500.000,APO_FAC 50.0000,AXIS_VEL 100.000,AXIS_ACC 100.000,ORI_TYP #VAR,CIRC_TYP #BASE,JERK_FAC 50.0000,GEAR_JERK 100.000,EXAX_IGN 0}
DECL E6POS XP3063={X 365.0,Y 368.0,Z -17.64,A -180,B 0,C 180,S 2,T 10,E1 0.0,E2 0.0,E3 0.0,E4 0.0,E5 0.0,E6 0.0}
DECL FDAT FP3063={TOOL_NO 1,BASE_NO 0,IPO_FRAME #BASE,POINT2[] " "}
DECL LDAT LCPDAT3063={VEL 2.00000,ACC 100.000,APO_DIST 500.000,APO_FAC 50.0000,AXIS_VEL 100.000,AXIS_ACC 100.000,ORI_TYP #VAR,CIRC_TYP #BASE,JERK_FAC 50.0000,GEAR_JERK 100.000,EXAX_IGN 0}
DECL E6POS XP3064={X 363.0,Y 370.0,Z -17.64,A -180,B 0,C 180,S 2,T 10,E1 0.0,E2 0.0,E3 0.0,E4 0.0,E5 0.0,E6 0.0}
DECL FDAT FP3064={TOOL_NO 1,BASE_NO 0,IPO_FRAME #BASE,POINT2[] " "}
DECL LDAT LCPDAT3064={VEL 2.00000,ACC 100.000,APO_DIST 500.000,APO_FAC 50.0000,AXIS_VEL 100.000,AXIS_ACC 100.000,ORI_TYP #VAR,CIRC_TYP #BASE,JERK_FAC 50.0000,GEAR_JERK 100.000,EXAX_IGN 0}
DECL E6POS XP3065={X 363.0,Y 370.0,Z -17.64,A -180,B 0,C 180,S 2,T 10,E1 0.0,E2 0.0,E3 0.0,E4 0.0,E5 0.0,E6 0.0}
DECL FDAT FP3065={TOOL_NO 1,BASE_NO 0,IPO_FRAME #BASE,POINT2[] " "}
DECL LDAT LCPDAT3065={VEL 2.00000,ACC 100.000,APO_DIST 500.000,APO_FAC 50.0000,AXIS_VEL 100.000,AXIS_ACC 100.000,ORI_TYP #VAR,CIRC_TYP #BASE,JERK_FAC 50.0000,GEAR_JERK 100.000,EXAX_IGN 0}
DECL E6POS XP3066={X 362.0,Y 370.0,Z -17.64,A -180,B 0,C 180,S 2,T 10,E1 0.0,E2 0.0,E3 0.0,E4 0.0,E5 0.0,E6 0.0}
DECL FDAT FP3066={TOOL_NO 1,BASE_NO 0,IPO_FRAME #BASE,POINT2[] " "}
DECL LDAT LCPDAT3066={VEL 2.00000,ACC 100.000,APO_DIST 500.000,APO_FAC 50.0000,AXIS_VEL 100.000,AXIS_ACC 100.000,ORI_TYP #VAR,CIRC_TYP #BASE,JERK_FAC 50.0000,GEAR_JERK 100.000,EXAX_IGN 0}
DECL E6POS XP3067={X 362.0,Y 370.0,Z -17.64,A -180,B 0,C 180,S 2,T 10,E1 0.0,E2 0.0,E3 0.0,E4 0.0,E5 0.0,E6 0.0}
DECL FDAT FP3067={TOOL_NO 1,BASE_NO 0,IPO_FRAME #BASE,POINT2[] " "}
DECL LDAT LCPDAT3067={VEL 2.00000,ACC 100.000,APO_DIST 500.000,APO_FAC 50.0000,AXIS_VEL 100.000,AXIS_ACC 100.000,ORI_TYP #VAR,CIRC_TYP #BASE,JERK_FAC 50.0000,GEAR_JERK 100.000,EXAX_IGN 0}
DECL E6POS XP3068={X 360.0,Y 372.0,Z -17.64,A -180,B 0,C 180,S 2,T 10,E1 0.0,E2 0.0,E3 0.0,E4 0.0,E5 0.0,E6 0.0}
DECL FDAT FP3068={TOOL_NO 1,BASE_NO 0,IPO_FRAME #BASE,POINT2[] " "}
DECL LDAT LCPDAT3068={VEL 2.00000,ACC 100.000,APO_DIST 500.000,APO_FAC 50.0000,AXIS_VEL 100.000,AXIS_ACC 100.000,ORI_TYP #VAR,CIRC_TYP #BASE,JERK_FAC 50.0000,GEAR_JERK 100.000,EXAX_IGN 0}
DECL E6POS XP3069={X 360.0,Y 372.0,Z -17.64,A -180,B 0,C 180,S 2,T 10,E1 0.0,E2 0.0,E3 0.0,E4 0.0,E5 0.0,E6 0.0}
DECL FDAT FP3069={TOOL_NO 1,BASE_NO 0,IPO_FRAME #BASE,POINT2[] " "}
DECL LDAT LCPDAT3069={VEL 2.00000,ACC 100.000,APO_DIST 500.000,APO_FAC 50.0000,AXIS_VEL 100.000,AXIS_ACC 100.000,ORI_TYP #VAR,CIRC_TYP #BASE,JERK_FAC 50.0000,GEAR_JERK 100.000,EXAX_IGN 0}
DECL E6POS XP3070={X 364.0,Y 370.0,Z -17.64,A -180,B 0,C 180,S 2,T 10,E1 0.0,E2 0.0,E3 0.0,E4 0.0,E5 0.0,E6 0.0}
DECL FDAT FP3070={TOOL_NO 1,BASE_NO 0,IPO_FRAME #BASE,POINT2[] " "}
DECL LDAT LCPDAT3070={VEL 2.00000,ACC 100.000,APO_DIST 500.000,APO_FAC 50.0000,AXIS_VEL 100.000,AXIS_ACC 100.000,ORI_TYP #VAR,CIRC_TYP #BASE,JERK_FAC 50.0000,GEAR_JERK 100.000,EXAX_IGN 0}
DECL E6POS XP3071={X 364.0,Y 370.0,Z -17.64,A -180,B 0,C 180,S 2,T 10,E1 0.0,E2 0.0,E3 0.0,E4 0.0,E5 0.0,E6 0.0}
DECL FDAT FP3071={TOOL_NO 1,BASE_NO 0,IPO_FRAME #BASE,POINT2[] " "}
DECL LDAT LCPDAT3071={VEL 2.00000,ACC 100.000,APO_DIST 500.000,APO_FAC 50.0000,AXIS_VEL 100.000,AXIS_ACC 100.000,ORI_TYP #VAR,CIRC_TYP #BASE,JERK_FAC 50.0000,GEAR_JERK 100.000,EXAX_IGN 0}
DECL E6POS XP3072={X 366.0,Y 372.0,Z -17.64,A -180,B 0,C 180,S 2,T 10,E1 0.0,E2 0.0,E3 0.0,E4 0.0,E5 0.0,E6 0.0}
DECL FDAT FP3072={TOOL_NO 1,BASE_NO 0,IPO_FRAME #BASE,POINT2[] " "}
DECL LDAT LCPDAT3072={VEL 2.00000,ACC 100.000,APO_DIST 500.000,APO_FAC 50.0000,AXIS_VEL 100.000,AXIS_ACC 100.000,ORI_TYP #VAR,CIRC_TYP #BASE,JERK_FAC 50.0000,GEAR_JERK 100.000,EXAX_IGN 0}
DECL E6POS XP3073={X 366.0,Y 372.0,Z -17.64,A -180,B 0,C 180,S 2,T 10,E1 0.0,E2 0.0,E3 0.0,E4 0.0,E5 0.0,E6 0.0}
DECL FDAT FP3073={TOOL_NO 1,BASE_NO 0,IPO_FRAME #BASE,POINT2[] " "}
DECL LDAT LCPDAT3073={VEL 2.00000,ACC 100.000,APO_DIST 500.000,APO_FAC 50.0000,AXIS_VEL 100.000,AXIS_ACC 100.000,ORI_TYP #VAR,CIRC_TYP #BASE,JERK_FAC 50.0000,GEAR_JERK 100.000,EXAX_IGN 0}
DECL E6POS XP3074={X 361.0,Y 376.0,Z -17.64,A -180,B 0,C 180,S 2,T 10,E1 0.0,E2 0.0,E3 0.0,E4 0.0,E5 0.0,E6 0.0}
DECL FDAT FP3074={TOOL_NO 1,BASE_NO 0,IPO_FRAME #BASE,POINT2[] " "}
DECL LDAT LCPDAT3074={VEL 2.00000,ACC 100.000,APO_DIST 500.000,APO_FAC 50.0000,AXIS_VEL 100.000,AXIS_ACC 100.000,ORI_TYP #VAR,CIRC_TYP #BASE,JERK_FAC 50.0000,GEAR_JERK 100.000,EXAX_IGN 0}
DECL E6POS XP3075={X 361.0,Y 376.0,Z -17.64,A -180,B 0,C 180,S 2,T 10,E1 0.0,E2 0.0,E3 0.0,E4 0.0,E5 0.0,E6 0.0}
DECL FDAT FP3075={TOOL_NO 1,BASE_NO 0,IPO_FRAME #BASE,POINT2[] " "}
DECL LDAT LCPDAT3075={VEL 2.00000,ACC 100.000,APO_DIST 500.000,APO_FAC 50.0000,AXIS_VEL 100.000,AXIS_ACC 100.000,ORI_TYP #VAR,CIRC_TYP #BASE,JERK_FAC 50.0000,GEAR_JERK 100.000,EXAX_IGN 0}
DECL E6POS XP3076={X 359.0,Y 376.0,Z -17.64,A -180,B 0,C 180,S 2,T 10,E1 0.0,E2 0.0,E3 0.0,E4 0.0,E5 0.0,E6 0.0}
DECL FDAT FP3076={TOOL_NO 1,BASE_NO 0,IPO_FRAME #BASE,POINT2[] " "}
DECL LDAT LCPDAT3076={VEL 2.00000,ACC 100.000,APO_DIST 500.000,APO_FAC 50.0000,AXIS_VEL 100.000,AXIS_ACC 100.000,ORI_TYP #VAR,CIRC_TYP #BASE,JERK_FAC 50.0000,GEAR_JERK 100.000,EXAX_IGN 0}
DECL E6POS XP3077={X 359.0,Y 376.0,Z -17.64,A -180,B 0,C 180,S 2,T 10,E1 0.0,E2 0.0,E3 0.0,E4 0.0,E5 0.0,E6 0.0}
DECL FDAT FP3077={TOOL_NO 1,BASE_NO 0,IPO_FRAME #BASE,POINT2[] " "}
DECL LDAT LCPDAT3077={VEL 2.00000,ACC 100.000,APO_DIST 500.000,APO_FAC 50.0000,AXIS_VEL 100.000,AXIS_ACC 100.000,ORI_TYP #VAR,CIRC_TYP #BASE,JERK_FAC 50.0000,GEAR_JERK 100.000,EXAX_IGN 0}
DECL E6POS XP3078={X 356.0,Y 374.0,Z -17.64,A -180,B 0,C 180,S 2,T 10,E1 0.0,E2 0.0,E3 0.0,E4 0.0,E5 0.0,E6 0.0}
DECL FDAT FP3078={TOOL_NO 1,BASE_NO 0,IPO_FRAME #BASE,POINT2[] " "}
DECL LDAT LCPDAT3078={VEL 2.00000,ACC 100.000,APO_DIST 500.000,APO_FAC 50.0000,AXIS_VEL 100.000,AXIS_ACC 100.000,ORI_TYP #VAR,CIRC_TYP #BASE,JERK_FAC 50.0000,GEAR_JERK 100.000,EXAX_IGN 0}
DECL E6POS XP3079={X 356.0,Y 374.0,Z -17.64,A -180,B 0,C 180,S 2,T 10,E1 0.0,E2 0.0,E3 0.0,E4 0.0,E5 0.0,E6 0.0}
DECL FDAT FP3079={TOOL_NO 1,BASE_NO 0,IPO_FRAME #BASE,POINT2[] " "}
DECL LDAT LCPDAT3079={VEL 2.00000,ACC 100.000,APO_DIST 500.000,APO_FAC 50.0000,AXIS_VEL 100.000,AXIS_ACC 100.000,ORI_TYP #VAR,CIRC_TYP #BASE,JERK_FAC 50.0000,GEAR_JERK 100.000,EXAX_IGN 0}
DECL E6POS XP3080={X 356.0,Y 376.0,Z -17.64,A -180,B 0,C 180,S 2,T 10,E1 0.0,E2 0.0,E3 0.0,E4 0.0,E5 0.0,E6 0.0}
DECL FDAT FP3080={TOOL_NO 1,BASE_NO 0,IPO_FRAME #BASE,POINT2[] " "}
DECL LDAT LCPDAT3080={VEL 2.00000,ACC 100.000,APO_DIST 500.000,APO_FAC 50.0000,AXIS_VEL 100.000,AXIS_ACC 100.000,ORI_TYP #VAR,CIRC_TYP #BASE,JERK_FAC 50.0000,GEAR_JERK 100.000,EXAX_IGN 0}
DECL E6POS XP3081={X 356.0,Y 376.0,Z -17.64,A -180,B 0,C 180,S 2,T 10,E1 0.0,E2 0.0,E3 0.0,E4 0.0,E5 0.0,E6 0.0}
DECL FDAT FP3081={TOOL_NO 1,BASE_NO 0,IPO_FRAME #BASE,POINT2[] " "}
DECL LDAT LCPDAT3081={VEL 2.00000,ACC 100.000,APO_DIST 500.000,APO_FAC 50.0000,AXIS_VEL 100.000,AXIS_ACC 100.000,ORI_TYP #VAR,CIRC_TYP #BASE,JERK_FAC 50.0000,GEAR_JERK 100.000,EXAX_IGN 0}
DECL E6POS XP3082={X 357.0,Y 374.0,Z -17.64,A -180,B 0,C 180,S 2,T 10,E1 0.0,E2 0.0,E3 0.0,E4 0.0,E5 0.0,E6 0.0}
DECL FDAT FP3082={TOOL_NO 1,BASE_NO 0,IPO_FRAME #BASE,POINT2[] " "}
DECL LDAT LCPDAT3082={VEL 2.00000,ACC 100.000,APO_DIST 500.000,APO_FAC 50.0000,AXIS_VEL 100.000,AXIS_ACC 100.000,ORI_TYP #VAR,CIRC_TYP #BASE,JERK_FAC 50.0000,GEAR_JERK 100.000,EXAX_IGN 0}
DECL E6POS XP3083={X 357.0,Y 374.0,Z -17.64,A -180,B 0,C 180,S 2,T 10,E1 0.0,E2 0.0,E3 0.0,E4 0.0,E5 0.0,E6 0.0}
DECL FDAT FP3083={TOOL_NO 1,BASE_NO 0,IPO_FRAME #BASE,POINT2[] " "}
DECL LDAT LCPDAT3083={VEL 2.00000,ACC 100.000,APO_DIST 500.000,APO_FAC 50.0000,AXIS_VEL 100.000,AXIS_ACC 100.000,ORI_TYP #VAR,CIRC_TYP #BASE,JERK_FAC 50.0000,GEAR_JERK 100.000,EXAX_IGN 0}
DECL E6POS XP3084={X 359.0,Y 376.0,Z -17.64,A -180,B 0,C 180,S 2,T 10,E1 0.0,E2 0.0,E3 0.0,E4 0.0,E5 0.0,E6 0.0}
DECL FDAT FP3084={TOOL_NO 1,BASE_NO 0,IPO_FRAME #BASE,POINT2[] " "}
DECL LDAT LCPDAT3084={VEL 2.00000,ACC 100.000,APO_DIST 500.000,APO_FAC 50.0000,AXIS_VEL 100.000,AXIS_ACC 100.000,ORI_TYP #VAR,CIRC_TYP #BASE,JERK_FAC 50.0000,GEAR_JERK 100.000,EXAX_IGN 0}
DECL E6POS XP3085={X 359.0,Y 376.0,Z -17.64,A -180,B 0,C 180,S 2,T 10,E1 0.0,E2 0.0,E3 0.0,E4 0.0,E5 0.0,E6 0.0}
DECL FDAT FP3085={TOOL_NO 1,BASE_NO 0,IPO_FRAME #BASE,POINT2[] " "}
DECL LDAT LCPDAT3085={VEL 2.00000,ACC 100.000,APO_DIST 500.000,APO_FAC 50.0000,AXIS_VEL 100.000,AXIS_ACC 100.000,ORI_TYP #VAR,CIRC_TYP #BASE,JERK_FAC 50.0000,GEAR_JERK 100.000,EXAX_IGN 0}
DECL E6POS XP3086={X 357.0,Y 378.0,Z -17.64,A -180,B 0,C 180,S 2,T 10,E1 0.0,E2 0.0,E3 0.0,E4 0.0,E5 0.0,E6 0.0}
DECL FDAT FP3086={TOOL_NO 1,BASE_NO 0,IPO_FRAME #BASE,POINT2[] " "}
DECL LDAT LCPDAT3086={VEL 2.00000,ACC 100.000,APO_DIST 500.000,APO_FAC 50.0000,AXIS_VEL 100.000,AXIS_ACC 100.000,ORI_TYP #VAR,CIRC_TYP #BASE,JERK_FAC 50.0000,GEAR_JERK 100.000,EXAX_IGN 0}
DECL E6POS XP3087={X 357.0,Y 378.0,Z -17.64,A -180,B 0,C 180,S 2,T 10,E1 0.0,E2 0.0,E3 0.0,E4 0.0,E5 0.0,E6 0.0}
DECL FDAT FP3087={TOOL_NO 1,BASE_NO 0,IPO_FRAME #BASE,POINT2[] " "}
DECL LDAT LCPDAT3087={VEL 2.00000,ACC 100.000,APO_DIST 500.000,APO_FAC 50.0000,AXIS_VEL 100.000,AXIS_ACC 100.000,ORI_TYP #VAR,CIRC_TYP #BASE,JERK_FAC 50.0000,GEAR_JERK 100.000,EXAX_IGN 0}
DECL E6POS XP3088={X 355.0,Y 379.0,Z -17.64,A -180,B 0,C 180,S 2,T 10,E1 0.0,E2 0.0,E3 0.0,E4 0.0,E5 0.0,E6 0.0}
DECL FDAT FP3088={TOOL_NO 1,BASE_NO 0,IPO_FRAME #BASE,POINT2[] " "}
DECL LDAT LCPDAT3088={VEL 2.00000,ACC 100.000,APO_DIST 500.000,APO_FAC 50.0000,AXIS_VEL 100.000,AXIS_ACC 100.000,ORI_TYP #VAR,CIRC_TYP #BASE,JERK_FAC 50.0000,GEAR_JERK 100.000,EXAX_IGN 0}
DECL E6POS XP3089={X 355.0,Y 379.0,Z -17.64,A -180,B 0,C 180,S 2,T 10,E1 0.0,E2 0.0,E3 0.0,E4 0.0,E5 0.0,E6 0.0}
DECL FDAT FP3089={TOOL_NO 1,BASE_NO 0,IPO_FRAME #BASE,POINT2[] " "}
DECL LDAT LCPDAT3089={VEL 2.00000,ACC 100.000,APO_DIST 500.000,APO_FAC 50.0000,AXIS_VEL 100.000,AXIS_ACC 100.000,ORI_TYP #VAR,CIRC_TYP #BASE,JERK_FAC 50.0000,GEAR_JERK 100.000,EXAX_IGN 0}
DECL E6POS XP3090={X 350.0,Y 380.0,Z -17.64,A -180,B 0,C 180,S 2,T 10,E1 0.0,E2 0.0,E3 0.0,E4 0.0,E5 0.0,E6 0.0}
DECL FDAT FP3090={TOOL_NO 1,BASE_NO 0,IPO_FRAME #BASE,POINT2[] " "}
DECL LDAT LCPDAT3090={VEL 2.00000,ACC 100.000,APO_DIST 500.000,APO_FAC 50.0000,AXIS_VEL 100.000,AXIS_ACC 100.000,ORI_TYP #VAR,CIRC_TYP #BASE,JERK_FAC 50.0000,GEAR_JERK 100.000,EXAX_IGN 0}
DECL E6POS XP3091={X 350.0,Y 380.0,Z -17.64,A -180,B 0,C 180,S 2,T 10,E1 0.0,E2 0.0,E3 0.0,E4 0.0,E5 0.0,E6 0.0}
DECL FDAT FP3091={TOOL_NO 1,BASE_NO 0,IPO_FRAME #BASE,POINT2[] " "}
DECL LDAT LCPDAT3091={VEL 2.00000,ACC 100.000,APO_DIST 500.000,APO_FAC 50.0000,AXIS_VEL 100.000,AXIS_ACC 100.000,ORI_TYP #VAR,CIRC_TYP #BASE,JERK_FAC 50.0000,GEAR_JERK 100.000,EXAX_IGN 0}
DECL E6POS XP3092={X 344.0,Y 380.0,Z -17.64,A -180,B 0,C 180,S 2,T 10,E1 0.0,E2 0.0,E3 0.0,E4 0.0,E5 0.0,E6 0.0}
DECL FDAT FP3092={TOOL_NO 1,BASE_NO 0,IPO_FRAME #BASE,POINT2[] " "}
DECL LDAT LCPDAT3092={VEL 2.00000,ACC 100.000,APO_DIST 500.000,APO_FAC 50.0000,AXIS_VEL 100.000,AXIS_ACC 100.000,ORI_TYP #VAR,CIRC_TYP #BASE,JERK_FAC 50.0000,GEAR_JERK 100.000,EXAX_IGN 0}
DECL E6POS XP3093={X 344.0,Y 380.0,Z -17.64,A -180,B 0,C 180,S 2,T 10,E1 0.0,E2 0.0,E3 0.0,E4 0.0,E5 0.0,E6 0.0}
DECL FDAT FP3093={TOOL_NO 1,BASE_NO 0,IPO_FRAME #BASE,POINT2[] " "}
DECL LDAT LCPDAT3093={VEL 2.00000,ACC 100.000,APO_DIST 500.000,APO_FAC 50.0000,AXIS_VEL 100.000,AXIS_ACC 100.000,ORI_TYP #VAR,CIRC_TYP #BASE,JERK_FAC 50.0000,GEAR_JERK 100.000,EXAX_IGN 0}
DECL E6POS XP3094={X 333.0,Y 380.0,Z -17.64,A -180,B 0,C 180,S 2,T 10,E1 0.0,E2 0.0,E3 0.0,E4 0.0,E5 0.0,E6 0.0}
DECL FDAT FP3094={TOOL_NO 1,BASE_NO 0,IPO_FRAME #BASE,POINT2[] " "}
DECL LDAT LCPDAT3094={VEL 2.00000,ACC 100.000,APO_DIST 500.000,APO_FAC 50.0000,AXIS_VEL 100.000,AXIS_ACC 100.000,ORI_TYP #VAR,CIRC_TYP #BASE,JERK_FAC 50.0000,GEAR_JERK 100.000,EXAX_IGN 0}
DECL E6POS XP3095={X 333.0,Y 380.0,Z -17.64,A -180,B 0,C 180,S 2,T 10,E1 0.0,E2 0.0,E3 0.0,E4 0.0,E5 0.0,E6 0.0}
DECL FDAT FP3095={TOOL_NO 1,BASE_NO 0,IPO_FRAME #BASE,POINT2[] " "}
DECL LDAT LCPDAT3095={VEL 2.00000,ACC 100.000,APO_DIST 500.000,APO_FAC 50.0000,AXIS_VEL 100.000,AXIS_ACC 100.000,ORI_TYP #VAR,CIRC_TYP #BASE,JERK_FAC 50.0000,GEAR_JERK 100.000,EXAX_IGN 0}
DECL E6POS XP3096={X 330.0,Y 379.0,Z -17.64,A -180,B 0,C 180,S 2,T 10,E1 0.0,E2 0.0,E3 0.0,E4 0.0,E5 0.0,E6 0.0}
DECL FDAT FP3096={TOOL_NO 1,BASE_NO 0,IPO_FRAME #BASE,POINT2[] " "}
DECL LDAT LCPDAT3096={VEL 2.00000,ACC 100.000,APO_DIST 500.000,APO_FAC 50.0000,AXIS_VEL 100.000,AXIS_ACC 100.000,ORI_TYP #VAR,CIRC_TYP #BASE,JERK_FAC 50.0000,GEAR_JERK 100.000,EXAX_IGN 0}
DECL E6POS XP3097={X 330.0,Y 379.0,Z -17.64,A -180,B 0,C 180,S 2,T 10,E1 0.0,E2 0.0,E3 0.0,E4 0.0,E5 0.0,E6 0.0}
DECL FDAT FP3097={TOOL_NO 1,BASE_NO 0,IPO_FRAME #BASE,POINT2[] " "}
DECL LDAT LCPDAT3097={VEL 2.00000,ACC 100.000,APO_DIST 500.000,APO_FAC 50.0000,AXIS_VEL 100.000,AXIS_ACC 100.000,ORI_TYP #VAR,CIRC_TYP #BASE,JERK_FAC 50.0000,GEAR_JERK 100.000,EXAX_IGN 0}
DECL E6POS XP3098={X 328.0,Y 378.0,Z -17.64,A -180,B 0,C 180,S 2,T 10,E1 0.0,E2 0.0,E3 0.0,E4 0.0,E5 0.0,E6 0.0}
DECL FDAT FP3098={TOOL_NO 1,BASE_NO 0,IPO_FRAME #BASE,POINT2[] " "}
DECL LDAT LCPDAT3098={VEL 2.00000,ACC 100.000,APO_DIST 500.000,APO_FAC 50.0000,AXIS_VEL 100.000,AXIS_ACC 100.000,ORI_TYP #VAR,CIRC_TYP #BASE,JERK_FAC 50.0000,GEAR_JERK 100.000,EXAX_IGN 0}
DECL E6POS XP3099={X 328.0,Y 378.0,Z -17.64,A -180,B 0,C 180,S 2,T 10,E1 0.0,E2 0.0,E3 0.0,E4 0.0,E5 0.0,E6 0.0}
DECL FDAT FP3099={TOOL_NO 1,BASE_NO 0,IPO_FRAME #BASE,POINT2[] " "}
DECL LDAT LCPDAT3099={VEL 2.00000,ACC 100.000,APO_DIST 500.000,APO_FAC 50.0000,AXIS_VEL 100.000,AXIS_ACC 100.000,ORI_TYP #VAR,CIRC_TYP #BASE,JERK_FAC 50.0000,GEAR_JERK 100.000,EXAX_IGN 0}
DECL E6POS XP3100={X 325.0,Y 375.0,Z -17.64,A -180,B 0,C 180,S 2,T 10,E1 0.0,E2 0.0,E3 0.0,E4 0.0,E5 0.0,E6 0.0}
DECL FDAT FP3100={TOOL_NO 1,BASE_NO 0,IPO_FRAME #BASE,POINT2[] " "}
DECL LDAT LCPDAT3100={VEL 2.00000,ACC 100.000,APO_DIST 500.000,APO_FAC 50.0000,AXIS_VEL 100.000,AXIS_ACC 100.000,ORI_TYP #VAR,CIRC_TYP #BASE,JERK_FAC 50.0000,GEAR_JERK 100.000,EXAX_IGN 0}
DECL E6POS XP3101={X 325.0,Y 375.0,Z -17.64,A -180,B 0,C 180,S 2,T 10,E1 0.0,E2 0.0,E3 0.0,E4 0.0,E5 0.0,E6 0.0}
DECL FDAT FP3101={TOOL_NO 1,BASE_NO 0,IPO_FRAME #BASE,POINT2[] " "}
DECL LDAT LCPDAT3101={VEL 2.00000,ACC 100.000,APO_DIST 500.000,APO_FAC 50.0000,AXIS_VEL 100.000,AXIS_ACC 100.000,ORI_TYP #VAR,CIRC_TYP #BASE,JERK_FAC 50.0000,GEAR_JERK 100.000,EXAX_IGN 0}
DECL E6POS XP3102={X 326.0,Y 373.0,Z -17.64,A -180,B 0,C 180,S 2,T 10,E1 0.0,E2 0.0,E3 0.0,E4 0.0,E5 0.0,E6 0.0}
DECL FDAT FP3102={TOOL_NO 1,BASE_NO 0,IPO_FRAME #BASE,POINT2[] " "}
DECL LDAT LCPDAT3102={VEL 2.00000,ACC 100.000,APO_DIST 500.000,APO_FAC 50.0000,AXIS_VEL 100.000,AXIS_ACC 100.000,ORI_TYP #VAR,CIRC_TYP #BASE,JERK_FAC 50.0000,GEAR_JERK 100.000,EXAX_IGN 0}
DECL E6POS XP3103={X 326.0,Y 373.0,Z -17.64,A -180,B 0,C 180,S 2,T 10,E1 0.0,E2 0.0,E3 0.0,E4 0.0,E5 0.0,E6 0.0}
DECL FDAT FP3103={TOOL_NO 1,BASE_NO 0,IPO_FRAME #BASE,POINT2[] " "}
DECL LDAT LCPDAT3103={VEL 2.00000,ACC 100.000,APO_DIST 500.000,APO_FAC 50.0000,AXIS_VEL 100.000,AXIS_ACC 100.000,ORI_TYP #VAR,CIRC_TYP #BASE,JERK_FAC 50.0000,GEAR_JERK 100.000,EXAX_IGN 0}
DECL E6POS XP3104={X 327.0,Y 371.0,Z -17.64,A -180,B 0,C 180,S 2,T 10,E1 0.0,E2 0.0,E3 0.0,E4 0.0,E5 0.0,E6 0.0}
DECL FDAT FP3104={TOOL_NO 1,BASE_NO 0,IPO_FRAME #BASE,POINT2[] " "}
DECL LDAT LCPDAT3104={VEL 2.00000,ACC 100.000,APO_DIST 500.000,APO_FAC 50.0000,AXIS_VEL 100.000,AXIS_ACC 100.000,ORI_TYP #VAR,CIRC_TYP #BASE,JERK_FAC 50.0000,GEAR_JERK 100.000,EXAX_IGN 0}
DECL E6POS XP3105={X 327.0,Y 371.0,Z -17.64,A -180,B 0,C 180,S 2,T 10,E1 0.0,E2 0.0,E3 0.0,E4 0.0,E5 0.0,E6 0.0}
DECL FDAT FP3105={TOOL_NO 1,BASE_NO 0,IPO_FRAME #BASE,POINT2[] " "}
DECL LDAT LCPDAT3105={VEL 2.00000,ACC 100.000,APO_DIST 500.000,APO_FAC 50.0000,AXIS_VEL 100.000,AXIS_ACC 100.000,ORI_TYP #VAR,CIRC_TYP #BASE,JERK_FAC 50.0000,GEAR_JERK 100.000,EXAX_IGN 0}
DECL E6POS XP3106={X 330.0,Y 368.0,Z -17.64,A -180,B 0,C 180,S 2,T 10,E1 0.0,E2 0.0,E3 0.0,E4 0.0,E5 0.0,E6 0.0}
DECL FDAT FP3106={TOOL_NO 1,BASE_NO 0,IPO_FRAME #BASE,POINT2[] " "}
DECL LDAT LCPDAT3106={VEL 2.00000,ACC 100.000,APO_DIST 500.000,APO_FAC 50.0000,AXIS_VEL 100.000,AXIS_ACC 100.000,ORI_TYP #VAR,CIRC_TYP #BASE,JERK_FAC 50.0000,GEAR_JERK 100.000,EXAX_IGN 0}
DECL E6POS XP3107={X 330.0,Y 368.0,Z -17.64,A -180,B 0,C 180,S 2,T 10,E1 0.0,E2 0.0,E3 0.0,E4 0.0,E5 0.0,E6 0.0}
DECL FDAT FP3107={TOOL_NO 1,BASE_NO 0,IPO_FRAME #BASE,POINT2[] " "}
DECL LDAT LCPDAT3107={VEL 2.00000,ACC 100.000,APO_DIST 500.000,APO_FAC 50.0000,AXIS_VEL 100.000,AXIS_ACC 100.000,ORI_TYP #VAR,CIRC_TYP #BASE,JERK_FAC 50.0000,GEAR_JERK 100.000,EXAX_IGN 0}
DECL E6POS XP3108={X 333.0,Y 366.0,Z -17.64,A -180,B 0,C 180,S 2,T 10,E1 0.0,E2 0.0,E3 0.0,E4 0.0,E5 0.0,E6 0.0}
DECL FDAT FP3108={TOOL_NO 1,BASE_NO 0,IPO_FRAME #BASE,POINT2[] " "}
DECL LDAT LCPDAT3108={VEL 2.00000,ACC 100.000,APO_DIST 500.000,APO_FAC 50.0000,AXIS_VEL 100.000,AXIS_ACC 100.000,ORI_TYP #VAR,CIRC_TYP #BASE,JERK_FAC 50.0000,GEAR_JERK 100.000,EXAX_IGN 0}
DECL E6POS XP3109={X 333.0,Y 366.0,Z -17.64,A -180,B 0,C 180,S 2,T 10,E1 0.0,E2 0.0,E3 0.0,E4 0.0,E5 0.0,E6 0.0}
DECL FDAT FP3109={TOOL_NO 1,BASE_NO 0,IPO_FRAME #BASE,POINT2[] " "}
DECL LDAT LCPDAT3109={VEL 2.00000,ACC 100.000,APO_DIST 500.000,APO_FAC 50.0000,AXIS_VEL 100.000,AXIS_ACC 100.000,ORI_TYP #VAR,CIRC_TYP #BASE,JERK_FAC 50.0000,GEAR_JERK 100.000,EXAX_IGN 0}
DECL E6POS XP3110={X 336.0,Y 365.0,Z -17.64,A -180,B 0,C 180,S 2,T 10,E1 0.0,E2 0.0,E3 0.0,E4 0.0,E5 0.0,E6 0.0}
DECL FDAT FP3110={TOOL_NO 1,BASE_NO 0,IPO_FRAME #BASE,POINT2[] " "}
DECL LDAT LCPDAT3110={VEL 2.00000,ACC 100.000,APO_DIST 500.000,APO_FAC 50.0000,AXIS_VEL 100.000,AXIS_ACC 100.000,ORI_TYP #VAR,CIRC_TYP #BASE,JERK_FAC 50.0000,GEAR_JERK 100.000,EXAX_IGN 0}
DECL E6POS XP3111={X 336.0,Y 365.0,Z -17.64,A -180,B 0,C 180,S 2,T 10,E1 0.0,E2 0.0,E3 0.0,E4 0.0,E5 0.0,E6 0.0}
DECL FDAT FP3111={TOOL_NO 1,BASE_NO 0,IPO_FRAME #BASE,POINT2[] " "}
DECL LDAT LCPDAT3111={VEL 2.00000,ACC 100.000,APO_DIST 500.000,APO_FAC 50.0000,AXIS_VEL 100.000,AXIS_ACC 100.000,ORI_TYP #VAR,CIRC_TYP #BASE,JERK_FAC 50.0000,GEAR_JERK 100.000,EXAX_IGN 0}
DECL E6POS XP3112={X 339.0,Y 366.0,Z -17.64,A -180,B 0,C 180,S 2,T 10,E1 0.0,E2 0.0,E3 0.0,E4 0.0,E5 0.0,E6 0.0}
DECL FDAT FP3112={TOOL_NO 1,BASE_NO 0,IPO_FRAME #BASE,POINT2[] " "}
DECL LDAT LCPDAT3112={VEL 2.00000,ACC 100.000,APO_DIST 500.000,APO_FAC 50.0000,AXIS_VEL 100.000,AXIS_ACC 100.000,ORI_TYP #VAR,CIRC_TYP #BASE,JERK_FAC 50.0000,GEAR_JERK 100.000,EXAX_IGN 0}
DECL E6POS XP3113={X 339.0,Y 366.0,Z -17.64,A -180,B 0,C 180,S 2,T 10,E1 0.0,E2 0.0,E3 0.0,E4 0.0,E5 0.0,E6 0.0}
DECL FDAT FP3113={TOOL_NO 1,BASE_NO 0,IPO_FRAME #BASE,POINT2[] " "}
DECL LDAT LCPDAT3113={VEL 2.00000,ACC 100.000,APO_DIST 500.000,APO_FAC 50.0000,AXIS_VEL 100.000,AXIS_ACC 100.000,ORI_TYP #VAR,CIRC_TYP #BASE,JERK_FAC 50.0000,GEAR_JERK 100.000,EXAX_IGN 0}
DECL E6POS XP3114={X 336.0,Y 367.0,Z -17.64,A -180,B 0,C 180,S 2,T 10,E1 0.0,E2 0.0,E3 0.0,E4 0.0,E5 0.0,E6 0.0}
DECL FDAT FP3114={TOOL_NO 1,BASE_NO 0,IPO_FRAME #BASE,POINT2[] " "}
DECL LDAT LCPDAT3114={VEL 2.00000,ACC 100.000,APO_DIST 500.000,APO_FAC 50.0000,AXIS_VEL 100.000,AXIS_ACC 100.000,ORI_TYP #VAR,CIRC_TYP #BASE,JERK_FAC 50.0000,GEAR_JERK 100.000,EXAX_IGN 0}
DECL E6POS XP3115={X 336.0,Y 367.0,Z -17.64,A -180,B 0,C 180,S 2,T 10,E1 0.0,E2 0.0,E3 0.0,E4 0.0,E5 0.0,E6 0.0}
DECL FDAT FP3115={TOOL_NO 1,BASE_NO 0,IPO_FRAME #BASE,POINT2[] " "}
DECL LDAT LCPDAT3115={VEL 2.00000,ACC 100.000,APO_DIST 500.000,APO_FAC 50.0000,AXIS_VEL 100.000,AXIS_ACC 100.000,ORI_TYP #VAR,CIRC_TYP #BASE,JERK_FAC 50.0000,GEAR_JERK 100.000,EXAX_IGN 0}
DECL E6POS XP3116={X 334.0,Y 369.0,Z -17.64,A -180,B 0,C 180,S 2,T 10,E1 0.0,E2 0.0,E3 0.0,E4 0.0,E5 0.0,E6 0.0}
DECL FDAT FP3116={TOOL_NO 1,BASE_NO 0,IPO_FRAME #BASE,POINT2[] " "}
DECL LDAT LCPDAT3116={VEL 2.00000,ACC 100.000,APO_DIST 500.000,APO_FAC 50.0000,AXIS_VEL 100.000,AXIS_ACC 100.000,ORI_TYP #VAR,CIRC_TYP #BASE,JERK_FAC 50.0000,GEAR_JERK 100.000,EXAX_IGN 0}
DECL E6POS XP3117={X 334.0,Y 369.0,Z -17.64,A -180,B 0,C 180,S 2,T 10,E1 0.0,E2 0.0,E3 0.0,E4 0.0,E5 0.0,E6 0.0}
DECL FDAT FP3117={TOOL_NO 1,BASE_NO 0,IPO_FRAME #BASE,POINT2[] " "}
DECL LDAT LCPDAT3117={VEL 2.00000,ACC 100.000,APO_DIST 500.000,APO_FAC 50.0000,AXIS_VEL 100.000,AXIS_ACC 100.000,ORI_TYP #VAR,CIRC_TYP #BASE,JERK_FAC 50.0000,GEAR_JERK 100.000,EXAX_IGN 0}
DECL E6POS XP3118={X 332.0,Y 370.0,Z -17.64,A -180,B 0,C 180,S 2,T 10,E1 0.0,E2 0.0,E3 0.0,E4 0.0,E5 0.0,E6 0.0}
DECL FDAT FP3118={TOOL_NO 1,BASE_NO 0,IPO_FRAME #BASE,POINT2[] " "}
DECL LDAT LCPDAT3118={VEL 2.00000,ACC 100.000,APO_DIST 500.000,APO_FAC 50.0000,AXIS_VEL 100.000,AXIS_ACC 100.000,ORI_TYP #VAR,CIRC_TYP #BASE,JERK_FAC 50.0000,GEAR_JERK 100.000,EXAX_IGN 0}
DECL E6POS XP3119={X 332.0,Y 370.0,Z -17.64,A -180,B 0,C 180,S 2,T 10,E1 0.0,E2 0.0,E3 0.0,E4 0.0,E5 0.0,E6 0.0}
DECL FDAT FP3119={TOOL_NO 1,BASE_NO 0,IPO_FRAME #BASE,POINT2[] " "}
DECL LDAT LCPDAT3119={VEL 2.00000,ACC 100.000,APO_DIST 500.000,APO_FAC 50.0000,AXIS_VEL 100.000,AXIS_ACC 100.000,ORI_TYP #VAR,CIRC_TYP #BASE,JERK_FAC 50.0000,GEAR_JERK 100.000,EXAX_IGN 0}
DECL E6POS XP3120={X 336.0,Y 367.0,Z -17.64,A -180,B 0,C 180,S 2,T 10,E1 0.0,E2 0.0,E3 0.0,E4 0.0,E5 0.0,E6 0.0}
DECL FDAT FP3120={TOOL_NO 1,BASE_NO 0,IPO_FRAME #BASE,POINT2[] " "}
DECL LDAT LCPDAT3120={VEL 2.00000,ACC 100.000,APO_DIST 500.000,APO_FAC 50.0000,AXIS_VEL 100.000,AXIS_ACC 100.000,ORI_TYP #VAR,CIRC_TYP #BASE,JERK_FAC 50.0000,GEAR_JERK 100.000,EXAX_IGN 0}
DECL E6POS XP3121={X 336.0,Y 367.0,Z -17.64,A -180,B 0,C 180,S 2,T 10,E1 0.0,E2 0.0,E3 0.0,E4 0.0,E5 0.0,E6 0.0}
DECL FDAT FP3121={TOOL_NO 1,BASE_NO 0,IPO_FRAME #BASE,POINT2[] " "}
DECL LDAT LCPDAT3121={VEL 2.00000,ACC 100.000,APO_DIST 500.000,APO_FAC 50.0000,AXIS_VEL 100.000,AXIS_ACC 100.000,ORI_TYP #VAR,CIRC_TYP #BASE,JERK_FAC 50.0000,GEAR_JERK 100.000,EXAX_IGN 0}
DECL E6POS XP3122={X 338.0,Y 366.0,Z -17.64,A -180,B 0,C 180,S 2,T 10,E1 0.0,E2 0.0,E3 0.0,E4 0.0,E5 0.0,E6 0.0}
DECL FDAT FP3122={TOOL_NO 1,BASE_NO 0,IPO_FRAME #BASE,POINT2[] " "}
DECL LDAT LCPDAT3122={VEL 2.00000,ACC 100.000,APO_DIST 500.000,APO_FAC 50.0000,AXIS_VEL 100.000,AXIS_ACC 100.000,ORI_TYP #VAR,CIRC_TYP #BASE,JERK_FAC 50.0000,GEAR_JERK 100.000,EXAX_IGN 0}
DECL E6POS XP3123={X 338.0,Y 366.0,Z -17.64,A -180,B 0,C 180,S 2,T 10,E1 0.0,E2 0.0,E3 0.0,E4 0.0,E5 0.0,E6 0.0}
DECL FDAT FP3123={TOOL_NO 1,BASE_NO 0,IPO_FRAME #BASE,POINT2[] " "}
DECL LDAT LCPDAT3123={VEL 2.00000,ACC 100.000,APO_DIST 500.000,APO_FAC 50.0000,AXIS_VEL 100.000,AXIS_ACC 100.000,ORI_TYP #VAR,CIRC_TYP #BASE,JERK_FAC 50.0000,GEAR_JERK 100.000,EXAX_IGN 0}
DECL E6POS XP3124={X 340.0,Y 365.0,Z -17.64,A -180,B 0,C 180,S 2,T 10,E1 0.0,E2 0.0,E3 0.0,E4 0.0,E5 0.0,E6 0.0}
DECL FDAT FP3124={TOOL_NO 1,BASE_NO 0,IPO_FRAME #BASE,POINT2[] " "}
DECL LDAT LCPDAT3124={VEL 2.00000,ACC 100.000,APO_DIST 500.000,APO_FAC 50.0000,AXIS_VEL 100.000,AXIS_ACC 100.000,ORI_TYP #VAR,CIRC_TYP #BASE,JERK_FAC 50.0000,GEAR_JERK 100.000,EXAX_IGN 0}
DECL E6POS XP3125={X 340.0,Y 365.0,Z -17.64,A -180,B 0,C 180,S 2,T 10,E1 0.0,E2 0.0,E3 0.0,E4 0.0,E5 0.0,E6 0.0}
DECL FDAT FP3125={TOOL_NO 1,BASE_NO 0,IPO_FRAME #BASE,POINT2[] " "}
DECL LDAT LCPDAT3125={VEL 2.00000,ACC 100.000,APO_DIST 500.000,APO_FAC 50.0000,AXIS_VEL 100.000,AXIS_ACC 100.000,ORI_TYP #VAR,CIRC_TYP #BASE,JERK_FAC 50.0000,GEAR_JERK 100.000,EXAX_IGN 0}
DECL E6POS XP3126={X 342.0,Y 364.0,Z -17.64,A -180,B 0,C 180,S 2,T 10,E1 0.0,E2 0.0,E3 0.0,E4 0.0,E5 0.0,E6 0.0}
DECL FDAT FP3126={TOOL_NO 1,BASE_NO 0,IPO_FRAME #BASE,POINT2[] " "}
DECL LDAT LCPDAT3126={VEL 2.00000,ACC 100.000,APO_DIST 500.000,APO_FAC 50.0000,AXIS_VEL 100.000,AXIS_ACC 100.000,ORI_TYP #VAR,CIRC_TYP #BASE,JERK_FAC 50.0000,GEAR_JERK 100.000,EXAX_IGN 0}
DECL E6POS XP3127={X 342.0,Y 364.0,Z -17.64,A -180,B 0,C 180,S 2,T 10,E1 0.0,E2 0.0,E3 0.0,E4 0.0,E5 0.0,E6 0.0}
DECL FDAT FP3127={TOOL_NO 1,BASE_NO 0,IPO_FRAME #BASE,POINT2[] " "}
DECL LDAT LCPDAT3127={VEL 2.00000,ACC 100.000,APO_DIST 500.000,APO_FAC 50.0000,AXIS_VEL 100.000,AXIS_ACC 100.000,ORI_TYP #VAR,CIRC_TYP #BASE,JERK_FAC 50.0000,GEAR_JERK 100.000,EXAX_IGN 0}
DECL E6POS XP3128={X 339.0,Y 363.0,Z -17.64,A -180,B 0,C 180,S 2,T 10,E1 0.0,E2 0.0,E3 0.0,E4 0.0,E5 0.0,E6 0.0}
DECL FDAT FP3128={TOOL_NO 1,BASE_NO 0,IPO_FRAME #BASE,POINT2[] " "}
DECL LDAT LCPDAT3128={VEL 2.00000,ACC 100.000,APO_DIST 500.000,APO_FAC 50.0000,AXIS_VEL 100.000,AXIS_ACC 100.000,ORI_TYP #VAR,CIRC_TYP #BASE,JERK_FAC 50.0000,GEAR_JERK 100.000,EXAX_IGN 0}
DECL E6POS XP3129={X 339.0,Y 363.0,Z -17.64,A -180,B 0,C 180,S 2,T 10,E1 0.0,E2 0.0,E3 0.0,E4 0.0,E5 0.0,E6 0.0}
DECL FDAT FP3129={TOOL_NO 1,BASE_NO 0,IPO_FRAME #BASE,POINT2[] " "}
DECL LDAT LCPDAT3129={VEL 2.00000,ACC 100.000,APO_DIST 500.000,APO_FAC 50.0000,AXIS_VEL 100.000,AXIS_ACC 100.000,ORI_TYP #VAR,CIRC_TYP #BASE,JERK_FAC 50.0000,GEAR_JERK 100.000,EXAX_IGN 0}
DECL E6POS XP3130={X 342.0,Y 362.0,Z -17.64,A -180,B 0,C 180,S 2,T 10,E1 0.0,E2 0.0,E3 0.0,E4 0.0,E5 0.0,E6 0.0}
DECL FDAT FP3130={TOOL_NO 1,BASE_NO 0,IPO_FRAME #BASE,POINT2[] " "}
DECL LDAT LCPDAT3130={VEL 2.00000,ACC 100.000,APO_DIST 500.000,APO_FAC 50.0000,AXIS_VEL 100.000,AXIS_ACC 100.000,ORI_TYP #VAR,CIRC_TYP #BASE,JERK_FAC 50.0000,GEAR_JERK 100.000,EXAX_IGN 0}
DECL E6POS XP3131={X 342.0,Y 362.0,Z -17.64,A -180,B 0,C 180,S 2,T 10,E1 0.0,E2 0.0,E3 0.0,E4 0.0,E5 0.0,E6 0.0}
DECL FDAT FP3131={TOOL_NO 1,BASE_NO 0,IPO_FRAME #BASE,POINT2[] " "}
DECL LDAT LCPDAT3131={VEL 2.00000,ACC 100.000,APO_DIST 500.000,APO_FAC 50.0000,AXIS_VEL 100.000,AXIS_ACC 100.000,ORI_TYP #VAR,CIRC_TYP #BASE,JERK_FAC 50.0000,GEAR_JERK 100.000,EXAX_IGN 0}
DECL E6POS XP3132={X 345.0,Y 359.0,Z -17.64,A -180,B 0,C 180,S 2,T 10,E1 0.0,E2 0.0,E3 0.0,E4 0.0,E5 0.0,E6 0.0}
DECL FDAT FP3132={TOOL_NO 1,BASE_NO 0,IPO_FRAME #BASE,POINT2[] " "}
DECL LDAT LCPDAT3132={VEL 2.00000,ACC 100.000,APO_DIST 500.000,APO_FAC 50.0000,AXIS_VEL 100.000,AXIS_ACC 100.000,ORI_TYP #VAR,CIRC_TYP #BASE,JERK_FAC 50.0000,GEAR_JERK 100.000,EXAX_IGN 0}
DECL E6POS XP3133={X 345.0,Y 359.0,Z -17.64,A -180,B 0,C 180,S 2,T 10,E1 0.0,E2 0.0,E3 0.0,E4 0.0,E5 0.0,E6 0.0}
DECL FDAT FP3133={TOOL_NO 1,BASE_NO 0,IPO_FRAME #BASE,POINT2[] " "}
DECL LDAT LCPDAT3133={VEL 2.00000,ACC 100.000,APO_DIST 500.000,APO_FAC 50.0000,AXIS_VEL 100.000,AXIS_ACC 100.000,ORI_TYP #VAR,CIRC_TYP #BASE,JERK_FAC 50.0000,GEAR_JERK 100.000,EXAX_IGN 0}
DECL E6POS XP3134={X 345.0,Y 354.0,Z -17.64,A -180,B 0,C 180,S 2,T 10,E1 0.0,E2 0.0,E3 0.0,E4 0.0,E5 0.0,E6 0.0}
DECL FDAT FP3134={TOOL_NO 1,BASE_NO 0,IPO_FRAME #BASE,POINT2[] " "}
DECL LDAT LCPDAT3134={VEL 2.00000,ACC 100.000,APO_DIST 500.000,APO_FAC 50.0000,AXIS_VEL 100.000,AXIS_ACC 100.000,ORI_TYP #VAR,CIRC_TYP #BASE,JERK_FAC 50.0000,GEAR_JERK 100.000,EXAX_IGN 0}
DECL E6POS XP3135={X 345.0,Y 354.0,Z -17.64,A -180,B 0,C 180,S 2,T 10,E1 0.0,E2 0.0,E3 0.0,E4 0.0,E5 0.0,E6 0.0}
DECL FDAT FP3135={TOOL_NO 1,BASE_NO 0,IPO_FRAME #BASE,POINT2[] " "}
DECL LDAT LCPDAT3135={VEL 2.00000,ACC 100.000,APO_DIST 500.000,APO_FAC 50.0000,AXIS_VEL 100.000,AXIS_ACC 100.000,ORI_TYP #VAR,CIRC_TYP #BASE,JERK_FAC 50.0000,GEAR_JERK 100.000,EXAX_IGN 0}
DECL E6POS XP3136={X 343.0,Y 353.0,Z -17.64,A -180,B 0,C 180,S 2,T 10,E1 0.0,E2 0.0,E3 0.0,E4 0.0,E5 0.0,E6 0.0}
DECL FDAT FP3136={TOOL_NO 1,BASE_NO 0,IPO_FRAME #BASE,POINT2[] " "}
DECL LDAT LCPDAT3136={VEL 2.00000,ACC 100.000,APO_DIST 500.000,APO_FAC 50.0000,AXIS_VEL 100.000,AXIS_ACC 100.000,ORI_TYP #VAR,CIRC_TYP #BASE,JERK_FAC 50.0000,GEAR_JERK 100.000,EXAX_IGN 0}
DECL E6POS XP3137={X 343.0,Y 353.0,Z -17.64,A -180,B 0,C 180,S 2,T 10,E1 0.0,E2 0.0,E3 0.0,E4 0.0,E5 0.0,E6 0.0}
DECL FDAT FP3137={TOOL_NO 1,BASE_NO 0,IPO_FRAME #BASE,POINT2[] " "}
DECL LDAT LCPDAT3137={VEL 2.00000,ACC 100.000,APO_DIST 500.000,APO_FAC 50.0000,AXIS_VEL 100.000,AXIS_ACC 100.000,ORI_TYP #VAR,CIRC_TYP #BASE,JERK_FAC 50.0000,GEAR_JERK 100.000,EXAX_IGN 0}
DECL E6POS XP3138={X 343.0,Y 351.0,Z -17.64,A -180,B 0,C 180,S 2,T 10,E1 0.0,E2 0.0,E3 0.0,E4 0.0,E5 0.0,E6 0.0}
DECL FDAT FP3138={TOOL_NO 1,BASE_NO 0,IPO_FRAME #BASE,POINT2[] " "}
DECL LDAT LCPDAT3138={VEL 2.00000,ACC 100.000,APO_DIST 500.000,APO_FAC 50.0000,AXIS_VEL 100.000,AXIS_ACC 100.000,ORI_TYP #VAR,CIRC_TYP #BASE,JERK_FAC 50.0000,GEAR_JERK 100.000,EXAX_IGN 0}
DECL E6POS XP3139={X 343.0,Y 351.0,Z -17.64,A -180,B 0,C 180,S 2,T 10,E1 0.0,E2 0.0,E3 0.0,E4 0.0,E5 0.0,E6 0.0}
DECL FDAT FP3139={TOOL_NO 1,BASE_NO 0,IPO_FRAME #BASE,POINT2[] " "}
DECL LDAT LCPDAT3139={VEL 2.00000,ACC 100.000,APO_DIST 500.000,APO_FAC 50.0000,AXIS_VEL 100.000,AXIS_ACC 100.000,ORI_TYP #VAR,CIRC_TYP #BASE,JERK_FAC 50.0000,GEAR_JERK 100.000,EXAX_IGN 0}
DECL E6POS XP3140={X 341.0,Y 349.0,Z -17.64,A -180,B 0,C 180,S 2,T 10,E1 0.0,E2 0.0,E3 0.0,E4 0.0,E5 0.0,E6 0.0}
DECL FDAT FP3140={TOOL_NO 1,BASE_NO 0,IPO_FRAME #BASE,POINT2[] " "}
DECL LDAT LCPDAT3140={VEL 2.00000,ACC 100.000,APO_DIST 500.000,APO_FAC 50.0000,AXIS_VEL 100.000,AXIS_ACC 100.000,ORI_TYP #VAR,CIRC_TYP #BASE,JERK_FAC 50.0000,GEAR_JERK 100.000,EXAX_IGN 0}
DECL E6POS XP3141={X 341.0,Y 349.0,Z -17.64,A -180,B 0,C 180,S 2,T 10,E1 0.0,E2 0.0,E3 0.0,E4 0.0,E5 0.0,E6 0.0}
DECL FDAT FP3141={TOOL_NO 1,BASE_NO 0,IPO_FRAME #BASE,POINT2[] " "}
DECL LDAT LCPDAT3141={VEL 2.00000,ACC 100.000,APO_DIST 500.000,APO_FAC 50.0000,AXIS_VEL 100.000,AXIS_ACC 100.000,ORI_TYP #VAR,CIRC_TYP #BASE,JERK_FAC 50.0000,GEAR_JERK 100.000,EXAX_IGN 0}
DECL E6POS XP3142={X 341.0,Y 348.0,Z -17.64,A -180,B 0,C 180,S 2,T 10,E1 0.0,E2 0.0,E3 0.0,E4 0.0,E5 0.0,E6 0.0}
DECL FDAT FP3142={TOOL_NO 1,BASE_NO 0,IPO_FRAME #BASE,POINT2[] " "}
DECL LDAT LCPDAT3142={VEL 2.00000,ACC 100.000,APO_DIST 500.000,APO_FAC 50.0000,AXIS_VEL 100.000,AXIS_ACC 100.000,ORI_TYP #VAR,CIRC_TYP #BASE,JERK_FAC 50.0000,GEAR_JERK 100.000,EXAX_IGN 0}
DECL E6POS XP3143={X 341.0,Y 348.0,Z -17.64,A -180,B 0,C 180,S 2,T 10,E1 0.0,E2 0.0,E3 0.0,E4 0.0,E5 0.0,E6 0.0}
DECL FDAT FP3143={TOOL_NO 1,BASE_NO 0,IPO_FRAME #BASE,POINT2[] " "}
DECL LDAT LCPDAT3143={VEL 2.00000,ACC 100.000,APO_DIST 500.000,APO_FAC 50.0000,AXIS_VEL 100.000,AXIS_ACC 100.000,ORI_TYP #VAR,CIRC_TYP #BASE,JERK_FAC 50.0000,GEAR_JERK 100.000,EXAX_IGN 0}
DECL E6POS XP3144={X 337.0,Y 347.0,Z -17.64,A -180,B 0,C 180,S 2,T 10,E1 0.0,E2 0.0,E3 0.0,E4 0.0,E5 0.0,E6 0.0}
DECL FDAT FP3144={TOOL_NO 1,BASE_NO 0,IPO_FRAME #BASE,POINT2[] " "}
DECL LDAT LCPDAT3144={VEL 2.00000,ACC 100.000,APO_DIST 500.000,APO_FAC 50.0000,AXIS_VEL 100.000,AXIS_ACC 100.000,ORI_TYP #VAR,CIRC_TYP #BASE,JERK_FAC 50.0000,GEAR_JERK 100.000,EXAX_IGN 0}
DECL E6POS XP3145={X 337.0,Y 347.0,Z -17.64,A -180,B 0,C 180,S 2,T 10,E1 0.0,E2 0.0,E3 0.0,E4 0.0,E5 0.0,E6 0.0}
DECL FDAT FP3145={TOOL_NO 1,BASE_NO 0,IPO_FRAME #BASE,POINT2[] " "}
DECL LDAT LCPDAT3145={VEL 2.00000,ACC 100.000,APO_DIST 500.000,APO_FAC 50.0000,AXIS_VEL 100.000,AXIS_ACC 100.000,ORI_TYP #VAR,CIRC_TYP #BASE,JERK_FAC 50.0000,GEAR_JERK 100.000,EXAX_IGN 0}
DECL E6POS XP3146={X 338.0,Y 351.0,Z -17.64,A -180,B 0,C 180,S 2,T 10,E1 0.0,E2 0.0,E3 0.0,E4 0.0,E5 0.0,E6 0.0}
DECL FDAT FP3146={TOOL_NO 1,BASE_NO 0,IPO_FRAME #BASE,POINT2[] " "}
DECL LDAT LCPDAT3146={VEL 2.00000,ACC 100.000,APO_DIST 500.000,APO_FAC 50.0000,AXIS_VEL 100.000,AXIS_ACC 100.000,ORI_TYP #VAR,CIRC_TYP #BASE,JERK_FAC 50.0000,GEAR_JERK 100.000,EXAX_IGN 0}
DECL E6POS XP3147={X 338.0,Y 351.0,Z -17.64,A -180,B 0,C 180,S 2,T 10,E1 0.0,E2 0.0,E3 0.0,E4 0.0,E5 0.0,E6 0.0}
DECL FDAT FP3147={TOOL_NO 1,BASE_NO 0,IPO_FRAME #BASE,POINT2[] " "}
DECL LDAT LCPDAT3147={VEL 2.00000,ACC 100.000,APO_DIST 500.000,APO_FAC 50.0000,AXIS_VEL 100.000,AXIS_ACC 100.000,ORI_TYP #VAR,CIRC_TYP #BASE,JERK_FAC 50.0000,GEAR_JERK 100.000,EXAX_IGN 0}
DECL E6POS XP3148={X 336.0,Y 355.0,Z -17.64,A -180,B 0,C 180,S 2,T 10,E1 0.0,E2 0.0,E3 0.0,E4 0.0,E5 0.0,E6 0.0}
DECL FDAT FP3148={TOOL_NO 1,BASE_NO 0,IPO_FRAME #BASE,POINT2[] " "}
DECL LDAT LCPDAT3148={VEL 2.00000,ACC 100.000,APO_DIST 500.000,APO_FAC 50.0000,AXIS_VEL 100.000,AXIS_ACC 100.000,ORI_TYP #VAR,CIRC_TYP #BASE,JERK_FAC 50.0000,GEAR_JERK 100.000,EXAX_IGN 0}
DECL E6POS XP3149={X 336.0,Y 355.0,Z -17.64,A -180,B 0,C 180,S 2,T 10,E1 0.0,E2 0.0,E3 0.0,E4 0.0,E5 0.0,E6 0.0}
DECL FDAT FP3149={TOOL_NO 1,BASE_NO 0,IPO_FRAME #BASE,POINT2[] " "}
DECL LDAT LCPDAT3149={VEL 2.00000,ACC 100.000,APO_DIST 500.000,APO_FAC 50.0000,AXIS_VEL 100.000,AXIS_ACC 100.000,ORI_TYP #VAR,CIRC_TYP #BASE,JERK_FAC 50.0000,GEAR_JERK 100.000,EXAX_IGN 0}
DECL E6POS XP3150={X 334.0,Y 354.0,Z -17.64,A -180,B 0,C 180,S 2,T 10,E1 0.0,E2 0.0,E3 0.0,E4 0.0,E5 0.0,E6 0.0}
DECL FDAT FP3150={TOOL_NO 1,BASE_NO 0,IPO_FRAME #BASE,POINT2[] " "}
DECL LDAT LCPDAT3150={VEL 2.00000,ACC 100.000,APO_DIST 500.000,APO_FAC 50.0000,AXIS_VEL 100.000,AXIS_ACC 100.000,ORI_TYP #VAR,CIRC_TYP #BASE,JERK_FAC 50.0000,GEAR_JERK 100.000,EXAX_IGN 0}
DECL E6POS XP3151={X 334.0,Y 354.0,Z -17.64,A -180,B 0,C 180,S 2,T 10,E1 0.0,E2 0.0,E3 0.0,E4 0.0,E5 0.0,E6 0.0}
DECL FDAT FP3151={TOOL_NO 1,BASE_NO 0,IPO_FRAME #BASE,POINT2[] " "}
DECL LDAT LCPDAT3151={VEL 2.00000,ACC 100.000,APO_DIST 500.000,APO_FAC 50.0000,AXIS_VEL 100.000,AXIS_ACC 100.000,ORI_TYP #VAR,CIRC_TYP #BASE,JERK_FAC 50.0000,GEAR_JERK 100.000,EXAX_IGN 0}
DECL E6POS XP3152={X 331.0,Y 347.0,Z -17.64,A -180,B 0,C 180,S 2,T 10,E1 0.0,E2 0.0,E3 0.0,E4 0.0,E5 0.0,E6 0.0}
DECL FDAT FP3152={TOOL_NO 1,BASE_NO 0,IPO_FRAME #BASE,POINT2[] " "}
DECL LDAT LCPDAT3152={VEL 2.00000,ACC 100.000,APO_DIST 500.000,APO_FAC 50.0000,AXIS_VEL 100.000,AXIS_ACC 100.000,ORI_TYP #VAR,CIRC_TYP #BASE,JERK_FAC 50.0000,GEAR_JERK 100.000,EXAX_IGN 0}
DECL E6POS XP3153={X 331.0,Y 347.0,Z -17.64,A -180,B 0,C 180,S 2,T 10,E1 0.0,E2 0.0,E3 0.0,E4 0.0,E5 0.0,E6 0.0}
DECL FDAT FP3153={TOOL_NO 1,BASE_NO 0,IPO_FRAME #BASE,POINT2[] " "}
DECL LDAT LCPDAT3153={VEL 2.00000,ACC 100.000,APO_DIST 500.000,APO_FAC 50.0000,AXIS_VEL 100.000,AXIS_ACC 100.000,ORI_TYP #VAR,CIRC_TYP #BASE,JERK_FAC 50.0000,GEAR_JERK 100.000,EXAX_IGN 0}
DECL E6POS XP3154={X 330.0,Y 350.0,Z -17.64,A -180,B 0,C 180,S 2,T 10,E1 0.0,E2 0.0,E3 0.0,E4 0.0,E5 0.0,E6 0.0}
DECL FDAT FP3154={TOOL_NO 1,BASE_NO 0,IPO_FRAME #BASE,POINT2[] " "}
DECL LDAT LCPDAT3154={VEL 2.00000,ACC 100.000,APO_DIST 500.000,APO_FAC 50.0000,AXIS_VEL 100.000,AXIS_ACC 100.000,ORI_TYP #VAR,CIRC_TYP #BASE,JERK_FAC 50.0000,GEAR_JERK 100.000,EXAX_IGN 0}
DECL E6POS XP3155={X 330.0,Y 350.0,Z -17.64,A -180,B 0,C 180,S 2,T 10,E1 0.0,E2 0.0,E3 0.0,E4 0.0,E5 0.0,E6 0.0}
DECL FDAT FP3155={TOOL_NO 1,BASE_NO 0,IPO_FRAME #BASE,POINT2[] " "}
DECL LDAT LCPDAT3155={VEL 2.00000,ACC 100.000,APO_DIST 500.000,APO_FAC 50.0000,AXIS_VEL 100.000,AXIS_ACC 100.000,ORI_TYP #VAR,CIRC_TYP #BASE,JERK_FAC 50.0000,GEAR_JERK 100.000,EXAX_IGN 0}
DECL E6POS XP3156={X 329.0,Y 348.0,Z -17.64,A -180,B 0,C 180,S 2,T 10,E1 0.0,E2 0.0,E3 0.0,E4 0.0,E5 0.0,E6 0.0}
DECL FDAT FP3156={TOOL_NO 1,BASE_NO 0,IPO_FRAME #BASE,POINT2[] " "}
DECL LDAT LCPDAT3156={VEL 2.00000,ACC 100.000,APO_DIST 500.000,APO_FAC 50.0000,AXIS_VEL 100.000,AXIS_ACC 100.000,ORI_TYP #VAR,CIRC_TYP #BASE,JERK_FAC 50.0000,GEAR_JERK 100.000,EXAX_IGN 0}
DECL E6POS XP3157={X 329.0,Y 348.0,Z -17.64,A -180,B 0,C 180,S 2,T 10,E1 0.0,E2 0.0,E3 0.0,E4 0.0,E5 0.0,E6 0.0}
DECL FDAT FP3157={TOOL_NO 1,BASE_NO 0,IPO_FRAME #BASE,POINT2[] " "}
DECL LDAT LCPDAT3157={VEL 2.00000,ACC 100.000,APO_DIST 500.000,APO_FAC 50.0000,AXIS_VEL 100.000,AXIS_ACC 100.000,ORI_TYP #VAR,CIRC_TYP #BASE,JERK_FAC 50.0000,GEAR_JERK 100.000,EXAX_IGN 0}
DECL E6POS XP3158={X 329.0,Y 345.0,Z -17.64,A -180,B 0,C 180,S 2,T 10,E1 0.0,E2 0.0,E3 0.0,E4 0.0,E5 0.0,E6 0.0}
DECL FDAT FP3158={TOOL_NO 1,BASE_NO 0,IPO_FRAME #BASE,POINT2[] " "}
DECL LDAT LCPDAT3158={VEL 2.00000,ACC 100.000,APO_DIST 500.000,APO_FAC 50.0000,AXIS_VEL 100.000,AXIS_ACC 100.000,ORI_TYP #VAR,CIRC_TYP #BASE,JERK_FAC 50.0000,GEAR_JERK 100.000,EXAX_IGN 0}
DECL E6POS XP3159={X 329.0,Y 345.0,Z -17.64,A -180,B 0,C 180,S 2,T 10,E1 0.0,E2 0.0,E3 0.0,E4 0.0,E5 0.0,E6 0.0}
DECL FDAT FP3159={TOOL_NO 1,BASE_NO 0,IPO_FRAME #BASE,POINT2[] " "}
DECL LDAT LCPDAT3159={VEL 2.00000,ACC 100.000,APO_DIST 500.000,APO_FAC 50.0000,AXIS_VEL 100.000,AXIS_ACC 100.000,ORI_TYP #VAR,CIRC_TYP #BASE,JERK_FAC 50.0000,GEAR_JERK 100.000,EXAX_IGN 0}
DECL E6POS XP3160={X 328.0,Y 342.0,Z -17.64,A -180,B 0,C 180,S 2,T 10,E1 0.0,E2 0.0,E3 0.0,E4 0.0,E5 0.0,E6 0.0}
DECL FDAT FP3160={TOOL_NO 1,BASE_NO 0,IPO_FRAME #BASE,POINT2[] " "}
DECL LDAT LCPDAT3160={VEL 2.00000,ACC 100.000,APO_DIST 500.000,APO_FAC 50.0000,AXIS_VEL 100.000,AXIS_ACC 100.000,ORI_TYP #VAR,CIRC_TYP #BASE,JERK_FAC 50.0000,GEAR_JERK 100.000,EXAX_IGN 0}
DECL E6POS XP3161={X 328.0,Y 342.0,Z -17.64,A -180,B 0,C 180,S 2,T 10,E1 0.0,E2 0.0,E3 0.0,E4 0.0,E5 0.0,E6 0.0}
DECL FDAT FP3161={TOOL_NO 1,BASE_NO 0,IPO_FRAME #BASE,POINT2[] " "}
DECL LDAT LCPDAT3161={VEL 2.00000,ACC 100.000,APO_DIST 500.000,APO_FAC 50.0000,AXIS_VEL 100.000,AXIS_ACC 100.000,ORI_TYP #VAR,CIRC_TYP #BASE,JERK_FAC 50.0000,GEAR_JERK 100.000,EXAX_IGN 0}
DECL E6POS XP3162={X 326.0,Y 338.0,Z -17.64,A -180,B 0,C 180,S 2,T 10,E1 0.0,E2 0.0,E3 0.0,E4 0.0,E5 0.0,E6 0.0}
DECL FDAT FP3162={TOOL_NO 1,BASE_NO 0,IPO_FRAME #BASE,POINT2[] " "}
DECL LDAT LCPDAT3162={VEL 2.00000,ACC 100.000,APO_DIST 500.000,APO_FAC 50.0000,AXIS_VEL 100.000,AXIS_ACC 100.000,ORI_TYP #VAR,CIRC_TYP #BASE,JERK_FAC 50.0000,GEAR_JERK 100.000,EXAX_IGN 0}
DECL E6POS XP3163={X 326.0,Y 338.0,Z -17.64,A -180,B 0,C 180,S 2,T 10,E1 0.0,E2 0.0,E3 0.0,E4 0.0,E5 0.0,E6 0.0}
DECL FDAT FP3163={TOOL_NO 1,BASE_NO 0,IPO_FRAME #BASE,POINT2[] " "}
DECL LDAT LCPDAT3163={VEL 2.00000,ACC 100.000,APO_DIST 500.000,APO_FAC 50.0000,AXIS_VEL 100.000,AXIS_ACC 100.000,ORI_TYP #VAR,CIRC_TYP #BASE,JERK_FAC 50.0000,GEAR_JERK 100.000,EXAX_IGN 0}
DECL E6POS XP3164={X 327.0,Y 334.0,Z -17.64,A -180,B 0,C 180,S 2,T 10,E1 0.0,E2 0.0,E3 0.0,E4 0.0,E5 0.0,E6 0.0}
DECL FDAT FP3164={TOOL_NO 1,BASE_NO 0,IPO_FRAME #BASE,POINT2[] " "}
DECL LDAT LCPDAT3164={VEL 2.00000,ACC 100.000,APO_DIST 500.000,APO_FAC 50.0000,AXIS_VEL 100.000,AXIS_ACC 100.000,ORI_TYP #VAR,CIRC_TYP #BASE,JERK_FAC 50.0000,GEAR_JERK 100.000,EXAX_IGN 0}
DECL E6POS XP3165={X 327.0,Y 334.0,Z -17.64,A -180,B 0,C 180,S 2,T 10,E1 0.0,E2 0.0,E3 0.0,E4 0.0,E5 0.0,E6 0.0}
DECL FDAT FP3165={TOOL_NO 1,BASE_NO 0,IPO_FRAME #BASE,POINT2[] " "}
DECL LDAT LCPDAT3165={VEL 2.00000,ACC 100.000,APO_DIST 500.000,APO_FAC 50.0000,AXIS_VEL 100.000,AXIS_ACC 100.000,ORI_TYP #VAR,CIRC_TYP #BASE,JERK_FAC 50.0000,GEAR_JERK 100.000,EXAX_IGN 0}
DECL E6POS XP3166={X 326.0,Y 332.0,Z -17.64,A -180,B 0,C 180,S 2,T 10,E1 0.0,E2 0.0,E3 0.0,E4 0.0,E5 0.0,E6 0.0}
DECL FDAT FP3166={TOOL_NO 1,BASE_NO 0,IPO_FRAME #BASE,POINT2[] " "}
DECL LDAT LCPDAT3166={VEL 2.00000,ACC 100.000,APO_DIST 500.000,APO_FAC 50.0000,AXIS_VEL 100.000,AXIS_ACC 100.000,ORI_TYP #VAR,CIRC_TYP #BASE,JERK_FAC 50.0000,GEAR_JERK 100.000,EXAX_IGN 0}
DECL E6POS XP3167={X 326.0,Y 332.0,Z -17.64,A -180,B 0,C 180,S 2,T 10,E1 0.0,E2 0.0,E3 0.0,E4 0.0,E5 0.0,E6 0.0}
DECL FDAT FP3167={TOOL_NO 1,BASE_NO 0,IPO_FRAME #BASE,POINT2[] " "}
DECL LDAT LCPDAT3167={VEL 2.00000,ACC 100.000,APO_DIST 500.000,APO_FAC 50.0000,AXIS_VEL 100.000,AXIS_ACC 100.000,ORI_TYP #VAR,CIRC_TYP #BASE,JERK_FAC 50.0000,GEAR_JERK 100.000,EXAX_IGN 0}
DECL E6POS XP3168={X 324.0,Y 330.0,Z -17.64,A -180,B 0,C 180,S 2,T 10,E1 0.0,E2 0.0,E3 0.0,E4 0.0,E5 0.0,E6 0.0}
DECL FDAT FP3168={TOOL_NO 1,BASE_NO 0,IPO_FRAME #BASE,POINT2[] " "}
DECL LDAT LCPDAT3168={VEL 2.00000,ACC 100.000,APO_DIST 500.000,APO_FAC 50.0000,AXIS_VEL 100.000,AXIS_ACC 100.000,ORI_TYP #VAR,CIRC_TYP #BASE,JERK_FAC 50.0000,GEAR_JERK 100.000,EXAX_IGN 0}
DECL E6POS XP3169={X 324.0,Y 330.0,Z -17.64,A -180,B 0,C 180,S 2,T 10,E1 0.0,E2 0.0,E3 0.0,E4 0.0,E5 0.0,E6 0.0}
DECL FDAT FP3169={TOOL_NO 1,BASE_NO 0,IPO_FRAME #BASE,POINT2[] " "}
DECL LDAT LCPDAT3169={VEL 2.00000,ACC 100.000,APO_DIST 500.000,APO_FAC 50.0000,AXIS_VEL 100.000,AXIS_ACC 100.000,ORI_TYP #VAR,CIRC_TYP #BASE,JERK_FAC 50.0000,GEAR_JERK 100.000,EXAX_IGN 0}
DECL E6POS XP3170={X 322.0,Y 330.0,Z -17.64,A -180,B 0,C 180,S 2,T 10,E1 0.0,E2 0.0,E3 0.0,E4 0.0,E5 0.0,E6 0.0}
DECL FDAT FP3170={TOOL_NO 1,BASE_NO 0,IPO_FRAME #BASE,POINT2[] " "}
DECL LDAT LCPDAT3170={VEL 2.00000,ACC 100.000,APO_DIST 500.000,APO_FAC 50.0000,AXIS_VEL 100.000,AXIS_ACC 100.000,ORI_TYP #VAR,CIRC_TYP #BASE,JERK_FAC 50.0000,GEAR_JERK 100.000,EXAX_IGN 0}
DECL E6POS XP3171={X 322.0,Y 330.0,Z -17.64,A -180,B 0,C 180,S 2,T 10,E1 0.0,E2 0.0,E3 0.0,E4 0.0,E5 0.0,E6 0.0}
DECL FDAT FP3171={TOOL_NO 1,BASE_NO 0,IPO_FRAME #BASE,POINT2[] " "}
DECL LDAT LCPDAT3171={VEL 2.00000,ACC 100.000,APO_DIST 500.000,APO_FAC 50.0000,AXIS_VEL 100.000,AXIS_ACC 100.000,ORI_TYP #VAR,CIRC_TYP #BASE,JERK_FAC 50.0000,GEAR_JERK 100.000,EXAX_IGN 0}
DECL E6POS XP3172={X 323.0,Y 336.0,Z -17.64,A -180,B 0,C 180,S 2,T 10,E1 0.0,E2 0.0,E3 0.0,E4 0.0,E5 0.0,E6 0.0}
DECL FDAT FP3172={TOOL_NO 1,BASE_NO 0,IPO_FRAME #BASE,POINT2[] " "}
DECL LDAT LCPDAT3172={VEL 2.00000,ACC 100.000,APO_DIST 500.000,APO_FAC 50.0000,AXIS_VEL 100.000,AXIS_ACC 100.000,ORI_TYP #VAR,CIRC_TYP #BASE,JERK_FAC 50.0000,GEAR_JERK 100.000,EXAX_IGN 0}
DECL E6POS XP3173={X 323.0,Y 336.0,Z -17.64,A -180,B 0,C 180,S 2,T 10,E1 0.0,E2 0.0,E3 0.0,E4 0.0,E5 0.0,E6 0.0}
DECL FDAT FP3173={TOOL_NO 1,BASE_NO 0,IPO_FRAME #BASE,POINT2[] " "}
DECL LDAT LCPDAT3173={VEL 2.00000,ACC 100.000,APO_DIST 500.000,APO_FAC 50.0000,AXIS_VEL 100.000,AXIS_ACC 100.000,ORI_TYP #VAR,CIRC_TYP #BASE,JERK_FAC 50.0000,GEAR_JERK 100.000,EXAX_IGN 0}
DECL E6POS XP3174={X 321.0,Y 336.0,Z -17.64,A -180,B 0,C 180,S 2,T 10,E1 0.0,E2 0.0,E3 0.0,E4 0.0,E5 0.0,E6 0.0}
DECL FDAT FP3174={TOOL_NO 1,BASE_NO 0,IPO_FRAME #BASE,POINT2[] " "}
DECL LDAT LCPDAT3174={VEL 2.00000,ACC 100.000,APO_DIST 500.000,APO_FAC 50.0000,AXIS_VEL 100.000,AXIS_ACC 100.000,ORI_TYP #VAR,CIRC_TYP #BASE,JERK_FAC 50.0000,GEAR_JERK 100.000,EXAX_IGN 0}
DECL E6POS XP3175={X 321.0,Y 336.0,Z -17.64,A -180,B 0,C 180,S 2,T 10,E1 0.0,E2 0.0,E3 0.0,E4 0.0,E5 0.0,E6 0.0}
DECL FDAT FP3175={TOOL_NO 1,BASE_NO 0,IPO_FRAME #BASE,POINT2[] " "}
DECL LDAT LCPDAT3175={VEL 2.00000,ACC 100.000,APO_DIST 500.000,APO_FAC 50.0000,AXIS_VEL 100.000,AXIS_ACC 100.000,ORI_TYP #VAR,CIRC_TYP #BASE,JERK_FAC 50.0000,GEAR_JERK 100.000,EXAX_IGN 0}
DECL E6POS XP3176={X 319.0,Y 336.0,Z -17.64,A -180,B 0,C 180,S 2,T 10,E1 0.0,E2 0.0,E3 0.0,E4 0.0,E5 0.0,E6 0.0}
DECL FDAT FP3176={TOOL_NO 1,BASE_NO 0,IPO_FRAME #BASE,POINT2[] " "}
DECL LDAT LCPDAT3176={VEL 2.00000,ACC 100.000,APO_DIST 500.000,APO_FAC 50.0000,AXIS_VEL 100.000,AXIS_ACC 100.000,ORI_TYP #VAR,CIRC_TYP #BASE,JERK_FAC 50.0000,GEAR_JERK 100.000,EXAX_IGN 0}
DECL E6POS XP3177={X 319.0,Y 336.0,Z -17.64,A -180,B 0,C 180,S 2,T 10,E1 0.0,E2 0.0,E3 0.0,E4 0.0,E5 0.0,E6 0.0}
DECL FDAT FP3177={TOOL_NO 1,BASE_NO 0,IPO_FRAME #BASE,POINT2[] " "}
DECL LDAT LCPDAT3177={VEL 2.00000,ACC 100.000,APO_DIST 500.000,APO_FAC 50.0000,AXIS_VEL 100.000,AXIS_ACC 100.000,ORI_TYP #VAR,CIRC_TYP #BASE,JERK_FAC 50.0000,GEAR_JERK 100.000,EXAX_IGN 0}
DECL E6POS XP3178={X 320.0,Y 334.0,Z -17.64,A -180,B 0,C 180,S 2,T 10,E1 0.0,E2 0.0,E3 0.0,E4 0.0,E5 0.0,E6 0.0}
DECL FDAT FP3178={TOOL_NO 1,BASE_NO 0,IPO_FRAME #BASE,POINT2[] " "}
DECL LDAT LCPDAT3178={VEL 2.00000,ACC 100.000,APO_DIST 500.000,APO_FAC 50.0000,AXIS_VEL 100.000,AXIS_ACC 100.000,ORI_TYP #VAR,CIRC_TYP #BASE,JERK_FAC 50.0000,GEAR_JERK 100.000,EXAX_IGN 0}
DECL E6POS XP3179={X 320.0,Y 334.0,Z -17.64,A -180,B 0,C 180,S 2,T 10,E1 0.0,E2 0.0,E3 0.0,E4 0.0,E5 0.0,E6 0.0}
DECL FDAT FP3179={TOOL_NO 1,BASE_NO 0,IPO_FRAME #BASE,POINT2[] " "}
DECL LDAT LCPDAT3179={VEL 2.00000,ACC 100.000,APO_DIST 500.000,APO_FAC 50.0000,AXIS_VEL 100.000,AXIS_ACC 100.000,ORI_TYP #VAR,CIRC_TYP #BASE,JERK_FAC 50.0000,GEAR_JERK 100.000,EXAX_IGN 0}
DECL E6POS XP3180={X 319.0,Y 331.0,Z -17.64,A -180,B 0,C 180,S 2,T 10,E1 0.0,E2 0.0,E3 0.0,E4 0.0,E5 0.0,E6 0.0}
DECL FDAT FP3180={TOOL_NO 1,BASE_NO 0,IPO_FRAME #BASE,POINT2[] " "}
DECL LDAT LCPDAT3180={VEL 2.00000,ACC 100.000,APO_DIST 500.000,APO_FAC 50.0000,AXIS_VEL 100.000,AXIS_ACC 100.000,ORI_TYP #VAR,CIRC_TYP #BASE,JERK_FAC 50.0000,GEAR_JERK 100.000,EXAX_IGN 0}
DECL E6POS XP3181={X 319.0,Y 331.0,Z -17.64,A -180,B 0,C 180,S 2,T 10,E1 0.0,E2 0.0,E3 0.0,E4 0.0,E5 0.0,E6 0.0}
DECL FDAT FP3181={TOOL_NO 1,BASE_NO 0,IPO_FRAME #BASE,POINT2[] " "}
DECL LDAT LCPDAT3181={VEL 2.00000,ACC 100.000,APO_DIST 500.000,APO_FAC 50.0000,AXIS_VEL 100.000,AXIS_ACC 100.000,ORI_TYP #VAR,CIRC_TYP #BASE,JERK_FAC 50.0000,GEAR_JERK 100.000,EXAX_IGN 0}
DECL E6POS XP3182={X 318.0,Y 329.0,Z -17.64,A -180,B 0,C 180,S 2,T 10,E1 0.0,E2 0.0,E3 0.0,E4 0.0,E5 0.0,E6 0.0}
DECL FDAT FP3182={TOOL_NO 1,BASE_NO 0,IPO_FRAME #BASE,POINT2[] " "}
DECL LDAT LCPDAT3182={VEL 2.00000,ACC 100.000,APO_DIST 500.000,APO_FAC 50.0000,AXIS_VEL 100.000,AXIS_ACC 100.000,ORI_TYP #VAR,CIRC_TYP #BASE,JERK_FAC 50.0000,GEAR_JERK 100.000,EXAX_IGN 0}
DECL E6POS XP3183={X 318.0,Y 329.0,Z -17.64,A -180,B 0,C 180,S 2,T 10,E1 0.0,E2 0.0,E3 0.0,E4 0.0,E5 0.0,E6 0.0}
DECL FDAT FP3183={TOOL_NO 1,BASE_NO 0,IPO_FRAME #BASE,POINT2[] " "}
DECL LDAT LCPDAT3183={VEL 2.00000,ACC 100.000,APO_DIST 500.000,APO_FAC 50.0000,AXIS_VEL 100.000,AXIS_ACC 100.000,ORI_TYP #VAR,CIRC_TYP #BASE,JERK_FAC 50.0000,GEAR_JERK 100.000,EXAX_IGN 0}
DECL E6POS XP3184={X 319.0,Y 331.0,Z -17.64,A -180,B 0,C 180,S 2,T 10,E1 0.0,E2 0.0,E3 0.0,E4 0.0,E5 0.0,E6 0.0}
DECL FDAT FP3184={TOOL_NO 1,BASE_NO 0,IPO_FRAME #BASE,POINT2[] " "}
DECL LDAT LCPDAT3184={VEL 2.00000,ACC 100.000,APO_DIST 500.000,APO_FAC 50.0000,AXIS_VEL 100.000,AXIS_ACC 100.000,ORI_TYP #VAR,CIRC_TYP #BASE,JERK_FAC 50.0000,GEAR_JERK 100.000,EXAX_IGN 0}
DECL E6POS XP3185={X 319.0,Y 331.0,Z -17.64,A -180,B 0,C 180,S 2,T 10,E1 0.0,E2 0.0,E3 0.0,E4 0.0,E5 0.0,E6 0.0}
DECL FDAT FP3185={TOOL_NO 1,BASE_NO 0,IPO_FRAME #BASE,POINT2[] " "}
DECL LDAT LCPDAT3185={VEL 2.00000,ACC 100.000,APO_DIST 500.000,APO_FAC 50.0000,AXIS_VEL 100.000,AXIS_ACC 100.000,ORI_TYP #VAR,CIRC_TYP #BASE,JERK_FAC 50.0000,GEAR_JERK 100.000,EXAX_IGN 0}
DECL E6POS XP3186={X 316.0,Y 331.0,Z -17.64,A -180,B 0,C 180,S 2,T 10,E1 0.0,E2 0.0,E3 0.0,E4 0.0,E5 0.0,E6 0.0}
DECL FDAT FP3186={TOOL_NO 1,BASE_NO 0,IPO_FRAME #BASE,POINT2[] " "}
DECL LDAT LCPDAT3186={VEL 2.00000,ACC 100.000,APO_DIST 500.000,APO_FAC 50.0000,AXIS_VEL 100.000,AXIS_ACC 100.000,ORI_TYP #VAR,CIRC_TYP #BASE,JERK_FAC 50.0000,GEAR_JERK 100.000,EXAX_IGN 0}
DECL E6POS XP3187={X 316.0,Y 331.0,Z -17.64,A -180,B 0,C 180,S 2,T 10,E1 0.0,E2 0.0,E3 0.0,E4 0.0,E5 0.0,E6 0.0}
DECL FDAT FP3187={TOOL_NO 1,BASE_NO 0,IPO_FRAME #BASE,POINT2[] " "}
DECL LDAT LCPDAT3187={VEL 2.00000,ACC 100.000,APO_DIST 500.000,APO_FAC 50.0000,AXIS_VEL 100.000,AXIS_ACC 100.000,ORI_TYP #VAR,CIRC_TYP #BASE,JERK_FAC 50.0000,GEAR_JERK 100.000,EXAX_IGN 0}
DECL E6POS XP3188={X 315.0,Y 329.0,Z -17.64,A -180,B 0,C 180,S 2,T 10,E1 0.0,E2 0.0,E3 0.0,E4 0.0,E5 0.0,E6 0.0}
DECL FDAT FP3188={TOOL_NO 1,BASE_NO 0,IPO_FRAME #BASE,POINT2[] " "}
DECL LDAT LCPDAT3188={VEL 2.00000,ACC 100.000,APO_DIST 500.000,APO_FAC 50.0000,AXIS_VEL 100.000,AXIS_ACC 100.000,ORI_TYP #VAR,CIRC_TYP #BASE,JERK_FAC 50.0000,GEAR_JERK 100.000,EXAX_IGN 0}
DECL E6POS XP3189={X 315.0,Y 329.0,Z -17.64,A -180,B 0,C 180,S 2,T 10,E1 0.0,E2 0.0,E3 0.0,E4 0.0,E5 0.0,E6 0.0}
DECL FDAT FP3189={TOOL_NO 1,BASE_NO 0,IPO_FRAME #BASE,POINT2[] " "}
DECL LDAT LCPDAT3189={VEL 2.00000,ACC 100.000,APO_DIST 500.000,APO_FAC 50.0000,AXIS_VEL 100.000,AXIS_ACC 100.000,ORI_TYP #VAR,CIRC_TYP #BASE,JERK_FAC 50.0000,GEAR_JERK 100.000,EXAX_IGN 0}
DECL E6POS XP3190={X 316.0,Y 326.0,Z -17.64,A -180,B 0,C 180,S 2,T 10,E1 0.0,E2 0.0,E3 0.0,E4 0.0,E5 0.0,E6 0.0}
DECL FDAT FP3190={TOOL_NO 1,BASE_NO 0,IPO_FRAME #BASE,POINT2[] " "}
DECL LDAT LCPDAT3190={VEL 2.00000,ACC 100.000,APO_DIST 500.000,APO_FAC 50.0000,AXIS_VEL 100.000,AXIS_ACC 100.000,ORI_TYP #VAR,CIRC_TYP #BASE,JERK_FAC 50.0000,GEAR_JERK 100.000,EXAX_IGN 0}
DECL E6POS XP3191={X 316.0,Y 326.0,Z -17.64,A -180,B 0,C 180,S 2,T 10,E1 0.0,E2 0.0,E3 0.0,E4 0.0,E5 0.0,E6 0.0}
DECL FDAT FP3191={TOOL_NO 1,BASE_NO 0,IPO_FRAME #BASE,POINT2[] " "}
DECL LDAT LCPDAT3191={VEL 2.00000,ACC 100.000,APO_DIST 500.000,APO_FAC 50.0000,AXIS_VEL 100.000,AXIS_ACC 100.000,ORI_TYP #VAR,CIRC_TYP #BASE,JERK_FAC 50.0000,GEAR_JERK 100.000,EXAX_IGN 0}
DECL E6POS XP3192={X 315.0,Y 329.0,Z -17.64,A -180,B 0,C 180,S 2,T 10,E1 0.0,E2 0.0,E3 0.0,E4 0.0,E5 0.0,E6 0.0}
DECL FDAT FP3192={TOOL_NO 1,BASE_NO 0,IPO_FRAME #BASE,POINT2[] " "}
DECL LDAT LCPDAT3192={VEL 2.00000,ACC 100.000,APO_DIST 500.000,APO_FAC 50.0000,AXIS_VEL 100.000,AXIS_ACC 100.000,ORI_TYP #VAR,CIRC_TYP #BASE,JERK_FAC 50.0000,GEAR_JERK 100.000,EXAX_IGN 0}
DECL E6POS XP3193={X 315.0,Y 329.0,Z -17.64,A -180,B 0,C 180,S 2,T 10,E1 0.0,E2 0.0,E3 0.0,E4 0.0,E5 0.0,E6 0.0}
DECL FDAT FP3193={TOOL_NO 1,BASE_NO 0,IPO_FRAME #BASE,POINT2[] " "}
DECL LDAT LCPDAT3193={VEL 2.00000,ACC 100.000,APO_DIST 500.000,APO_FAC 50.0000,AXIS_VEL 100.000,AXIS_ACC 100.000,ORI_TYP #VAR,CIRC_TYP #BASE,JERK_FAC 50.0000,GEAR_JERK 100.000,EXAX_IGN 0}
DECL E6POS XP3194={X 314.0,Y 327.0,Z -17.64,A -180,B 0,C 180,S 2,T 10,E1 0.0,E2 0.0,E3 0.0,E4 0.0,E5 0.0,E6 0.0}
DECL FDAT FP3194={TOOL_NO 1,BASE_NO 0,IPO_FRAME #BASE,POINT2[] " "}
DECL LDAT LCPDAT3194={VEL 2.00000,ACC 100.000,APO_DIST 500.000,APO_FAC 50.0000,AXIS_VEL 100.000,AXIS_ACC 100.000,ORI_TYP #VAR,CIRC_TYP #BASE,JERK_FAC 50.0000,GEAR_JERK 100.000,EXAX_IGN 0}
DECL E6POS XP3195={X 314.0,Y 327.0,Z -17.64,A -180,B 0,C 180,S 2,T 10,E1 0.0,E2 0.0,E3 0.0,E4 0.0,E5 0.0,E6 0.0}
DECL FDAT FP3195={TOOL_NO 1,BASE_NO 0,IPO_FRAME #BASE,POINT2[] " "}
DECL LDAT LCPDAT3195={VEL 2.00000,ACC 100.000,APO_DIST 500.000,APO_FAC 50.0000,AXIS_VEL 100.000,AXIS_ACC 100.000,ORI_TYP #VAR,CIRC_TYP #BASE,JERK_FAC 50.0000,GEAR_JERK 100.000,EXAX_IGN 0}
DECL E6POS XP3196={X 312.0,Y 328.0,Z -17.64,A -180,B 0,C 180,S 2,T 10,E1 0.0,E2 0.0,E3 0.0,E4 0.0,E5 0.0,E6 0.0}
DECL FDAT FP3196={TOOL_NO 1,BASE_NO 0,IPO_FRAME #BASE,POINT2[] " "}
DECL LDAT LCPDAT3196={VEL 2.00000,ACC 100.000,APO_DIST 500.000,APO_FAC 50.0000,AXIS_VEL 100.000,AXIS_ACC 100.000,ORI_TYP #VAR,CIRC_TYP #BASE,JERK_FAC 50.0000,GEAR_JERK 100.000,EXAX_IGN 0}
DECL E6POS XP3197={X 312.0,Y 328.0,Z -17.64,A -180,B 0,C 180,S 2,T 10,E1 0.0,E2 0.0,E3 0.0,E4 0.0,E5 0.0,E6 0.0}
DECL FDAT FP3197={TOOL_NO 1,BASE_NO 0,IPO_FRAME #BASE,POINT2[] " "}
DECL LDAT LCPDAT3197={VEL 2.00000,ACC 100.000,APO_DIST 500.000,APO_FAC 50.0000,AXIS_VEL 100.000,AXIS_ACC 100.000,ORI_TYP #VAR,CIRC_TYP #BASE,JERK_FAC 50.0000,GEAR_JERK 100.000,EXAX_IGN 0}
DECL E6POS XP3198={X 314.0,Y 328.0,Z -17.64,A -180,B 0,C 180,S 2,T 10,E1 0.0,E2 0.0,E3 0.0,E4 0.0,E5 0.0,E6 0.0}
DECL FDAT FP3198={TOOL_NO 1,BASE_NO 0,IPO_FRAME #BASE,POINT2[] " "}
DECL LDAT LCPDAT3198={VEL 2.00000,ACC 100.000,APO_DIST 500.000,APO_FAC 50.0000,AXIS_VEL 100.000,AXIS_ACC 100.000,ORI_TYP #VAR,CIRC_TYP #BASE,JERK_FAC 50.0000,GEAR_JERK 100.000,EXAX_IGN 0}
DECL E6POS XP3199={X 314.0,Y 328.0,Z -17.64,A -180,B 0,C 180,S 2,T 10,E1 0.0,E2 0.0,E3 0.0,E4 0.0,E5 0.0,E6 0.0}
DECL FDAT FP3199={TOOL_NO 1,BASE_NO 0,IPO_FRAME #BASE,POINT2[] " "}
DECL LDAT LCPDAT3199={VEL 2.00000,ACC 100.000,APO_DIST 500.000,APO_FAC 50.0000,AXIS_VEL 100.000,AXIS_ACC 100.000,ORI_TYP #VAR,CIRC_TYP #BASE,JERK_FAC 50.0000,GEAR_JERK 100.000,EXAX_IGN 0}
DECL E6POS XP3200={X 316.0,Y 331.0,Z -17.64,A -180,B 0,C 180,S 2,T 10,E1 0.0,E2 0.0,E3 0.0,E4 0.0,E5 0.0,E6 0.0}
DECL FDAT FP3200={TOOL_NO 1,BASE_NO 0,IPO_FRAME #BASE,POINT2[] " "}
DECL LDAT LCPDAT3200={VEL 2.00000,ACC 100.000,APO_DIST 500.000,APO_FAC 50.0000,AXIS_VEL 100.000,AXIS_ACC 100.000,ORI_TYP #VAR,CIRC_TYP #BASE,JERK_FAC 50.0000,GEAR_JERK 100.000,EXAX_IGN 0}
DECL E6POS XP3201={X 316.0,Y 331.0,Z -17.64,A -180,B 0,C 180,S 2,T 10,E1 0.0,E2 0.0,E3 0.0,E4 0.0,E5 0.0,E6 0.0}
DECL FDAT FP3201={TOOL_NO 1,BASE_NO 0,IPO_FRAME #BASE,POINT2[] " "}
DECL LDAT LCPDAT3201={VEL 2.00000,ACC 100.000,APO_DIST 500.000,APO_FAC 50.0000,AXIS_VEL 100.000,AXIS_ACC 100.000,ORI_TYP #VAR,CIRC_TYP #BASE,JERK_FAC 50.0000,GEAR_JERK 100.000,EXAX_IGN 0}
DECL E6POS XP3202={X 318.0,Y 336.0,Z -17.64,A -180,B 0,C 180,S 2,T 10,E1 0.0,E2 0.0,E3 0.0,E4 0.0,E5 0.0,E6 0.0}
DECL FDAT FP3202={TOOL_NO 1,BASE_NO 0,IPO_FRAME #BASE,POINT2[] " "}
DECL LDAT LCPDAT3202={VEL 2.00000,ACC 100.000,APO_DIST 500.000,APO_FAC 50.0000,AXIS_VEL 100.000,AXIS_ACC 100.000,ORI_TYP #VAR,CIRC_TYP #BASE,JERK_FAC 50.0000,GEAR_JERK 100.000,EXAX_IGN 0}
DECL E6POS XP3203={X 318.0,Y 336.0,Z -17.64,A -180,B 0,C 180,S 2,T 10,E1 0.0,E2 0.0,E3 0.0,E4 0.0,E5 0.0,E6 0.0}
DECL FDAT FP3203={TOOL_NO 1,BASE_NO 0,IPO_FRAME #BASE,POINT2[] " "}
DECL LDAT LCPDAT3203={VEL 2.00000,ACC 100.000,APO_DIST 500.000,APO_FAC 50.0000,AXIS_VEL 100.000,AXIS_ACC 100.000,ORI_TYP #VAR,CIRC_TYP #BASE,JERK_FAC 50.0000,GEAR_JERK 100.000,EXAX_IGN 0}
DECL E6POS XP3204={X 319.0,Y 336.0,Z -17.64,A -180,B 0,C 180,S 2,T 10,E1 0.0,E2 0.0,E3 0.0,E4 0.0,E5 0.0,E6 0.0}
DECL FDAT FP3204={TOOL_NO 1,BASE_NO 0,IPO_FRAME #BASE,POINT2[] " "}
DECL LDAT LCPDAT3204={VEL 2.00000,ACC 100.000,APO_DIST 500.000,APO_FAC 50.0000,AXIS_VEL 100.000,AXIS_ACC 100.000,ORI_TYP #VAR,CIRC_TYP #BASE,JERK_FAC 50.0000,GEAR_JERK 100.000,EXAX_IGN 0}
DECL E6POS XP3205={X 319.0,Y 336.0,Z -17.64,A -180,B 0,C 180,S 2,T 10,E1 0.0,E2 0.0,E3 0.0,E4 0.0,E5 0.0,E6 0.0}
DECL FDAT FP3205={TOOL_NO 1,BASE_NO 0,IPO_FRAME #BASE,POINT2[] " "}
DECL LDAT LCPDAT3205={VEL 2.00000,ACC 100.000,APO_DIST 500.000,APO_FAC 50.0000,AXIS_VEL 100.000,AXIS_ACC 100.000,ORI_TYP #VAR,CIRC_TYP #BASE,JERK_FAC 50.0000,GEAR_JERK 100.000,EXAX_IGN 0}
DECL E6POS XP3206={X 324.0,Y 337.0,Z -17.64,A -180,B 0,C 180,S 2,T 10,E1 0.0,E2 0.0,E3 0.0,E4 0.0,E5 0.0,E6 0.0}
DECL FDAT FP3206={TOOL_NO 1,BASE_NO 0,IPO_FRAME #BASE,POINT2[] " "}
DECL LDAT LCPDAT3206={VEL 2.00000,ACC 100.000,APO_DIST 500.000,APO_FAC 50.0000,AXIS_VEL 100.000,AXIS_ACC 100.000,ORI_TYP #VAR,CIRC_TYP #BASE,JERK_FAC 50.0000,GEAR_JERK 100.000,EXAX_IGN 0}
DECL E6POS XP3207={X 324.0,Y 337.0,Z -17.64,A -180,B 0,C 180,S 2,T 10,E1 0.0,E2 0.0,E3 0.0,E4 0.0,E5 0.0,E6 0.0}
DECL FDAT FP3207={TOOL_NO 1,BASE_NO 0,IPO_FRAME #BASE,POINT2[] " "}
DECL LDAT LCPDAT3207={VEL 2.00000,ACC 100.000,APO_DIST 500.000,APO_FAC 50.0000,AXIS_VEL 100.000,AXIS_ACC 100.000,ORI_TYP #VAR,CIRC_TYP #BASE,JERK_FAC 50.0000,GEAR_JERK 100.000,EXAX_IGN 0}
DECL E6POS XP3208={X 325.0,Y 338.0,Z -17.64,A -180,B 0,C 180,S 2,T 10,E1 0.0,E2 0.0,E3 0.0,E4 0.0,E5 0.0,E6 0.0}
DECL FDAT FP3208={TOOL_NO 1,BASE_NO 0,IPO_FRAME #BASE,POINT2[] " "}
DECL LDAT LCPDAT3208={VEL 2.00000,ACC 100.000,APO_DIST 500.000,APO_FAC 50.0000,AXIS_VEL 100.000,AXIS_ACC 100.000,ORI_TYP #VAR,CIRC_TYP #BASE,JERK_FAC 50.0000,GEAR_JERK 100.000,EXAX_IGN 0}
DECL E6POS XP3209={X 325.0,Y 338.0,Z -17.64,A -180,B 0,C 180,S 2,T 10,E1 0.0,E2 0.0,E3 0.0,E4 0.0,E5 0.0,E6 0.0}
DECL FDAT FP3209={TOOL_NO 1,BASE_NO 0,IPO_FRAME #BASE,POINT2[] " "}
DECL LDAT LCPDAT3209={VEL 2.00000,ACC 100.000,APO_DIST 500.000,APO_FAC 50.0000,AXIS_VEL 100.000,AXIS_ACC 100.000,ORI_TYP #VAR,CIRC_TYP #BASE,JERK_FAC 50.0000,GEAR_JERK 100.000,EXAX_IGN 0}
DECL E6POS XP3210={X 326.0,Y 339.0,Z -17.64,A -180,B 0,C 180,S 2,T 10,E1 0.0,E2 0.0,E3 0.0,E4 0.0,E5 0.0,E6 0.0}
DECL FDAT FP3210={TOOL_NO 1,BASE_NO 0,IPO_FRAME #BASE,POINT2[] " "}
DECL LDAT LCPDAT3210={VEL 2.00000,ACC 100.000,APO_DIST 500.000,APO_FAC 50.0000,AXIS_VEL 100.000,AXIS_ACC 100.000,ORI_TYP #VAR,CIRC_TYP #BASE,JERK_FAC 50.0000,GEAR_JERK 100.000,EXAX_IGN 0}
DECL E6POS XP3211={X 326.0,Y 339.0,Z -17.64,A -180,B 0,C 180,S 2,T 10,E1 0.0,E2 0.0,E3 0.0,E4 0.0,E5 0.0,E6 0.0}
DECL FDAT FP3211={TOOL_NO 1,BASE_NO 0,IPO_FRAME #BASE,POINT2[] " "}
DECL LDAT LCPDAT3211={VEL 2.00000,ACC 100.000,APO_DIST 500.000,APO_FAC 50.0000,AXIS_VEL 100.000,AXIS_ACC 100.000,ORI_TYP #VAR,CIRC_TYP #BASE,JERK_FAC 50.0000,GEAR_JERK 100.000,EXAX_IGN 0}
DECL E6POS XP3212={X 327.0,Y 341.0,Z -17.64,A -180,B 0,C 180,S 2,T 10,E1 0.0,E2 0.0,E3 0.0,E4 0.0,E5 0.0,E6 0.0}
DECL FDAT FP3212={TOOL_NO 1,BASE_NO 0,IPO_FRAME #BASE,POINT2[] " "}
DECL LDAT LCPDAT3212={VEL 2.00000,ACC 100.000,APO_DIST 500.000,APO_FAC 50.0000,AXIS_VEL 100.000,AXIS_ACC 100.000,ORI_TYP #VAR,CIRC_TYP #BASE,JERK_FAC 50.0000,GEAR_JERK 100.000,EXAX_IGN 0}
DECL E6POS XP3213={X 327.0,Y 341.0,Z -17.64,A -180,B 0,C 180,S 2,T 10,E1 0.0,E2 0.0,E3 0.0,E4 0.0,E5 0.0,E6 0.0}
DECL FDAT FP3213={TOOL_NO 1,BASE_NO 0,IPO_FRAME #BASE,POINT2[] " "}
DECL LDAT LCPDAT3213={VEL 2.00000,ACC 100.000,APO_DIST 500.000,APO_FAC 50.0000,AXIS_VEL 100.000,AXIS_ACC 100.000,ORI_TYP #VAR,CIRC_TYP #BASE,JERK_FAC 50.0000,GEAR_JERK 100.000,EXAX_IGN 0}
DECL E6POS XP3214={X 329.0,Y 345.0,Z -17.64,A -180,B 0,C 180,S 2,T 10,E1 0.0,E2 0.0,E3 0.0,E4 0.0,E5 0.0,E6 0.0}
DECL FDAT FP3214={TOOL_NO 1,BASE_NO 0,IPO_FRAME #BASE,POINT2[] " "}
DECL LDAT LCPDAT3214={VEL 2.00000,ACC 100.000,APO_DIST 500.000,APO_FAC 50.0000,AXIS_VEL 100.000,AXIS_ACC 100.000,ORI_TYP #VAR,CIRC_TYP #BASE,JERK_FAC 50.0000,GEAR_JERK 100.000,EXAX_IGN 0}
DECL E6POS XP3215={X 329.0,Y 345.0,Z -17.64,A -180,B 0,C 180,S 2,T 10,E1 0.0,E2 0.0,E3 0.0,E4 0.0,E5 0.0,E6 0.0}
DECL FDAT FP3215={TOOL_NO 1,BASE_NO 0,IPO_FRAME #BASE,POINT2[] " "}
DECL LDAT LCPDAT3215={VEL 2.00000,ACC 100.000,APO_DIST 500.000,APO_FAC 50.0000,AXIS_VEL 100.000,AXIS_ACC 100.000,ORI_TYP #VAR,CIRC_TYP #BASE,JERK_FAC 50.0000,GEAR_JERK 100.000,EXAX_IGN 0}
DECL E6POS XP3216={X 328.0,Y 348.0,Z -17.64,A -180,B 0,C 180,S 2,T 10,E1 0.0,E2 0.0,E3 0.0,E4 0.0,E5 0.0,E6 0.0}
DECL FDAT FP3216={TOOL_NO 1,BASE_NO 0,IPO_FRAME #BASE,POINT2[] " "}
DECL LDAT LCPDAT3216={VEL 2.00000,ACC 100.000,APO_DIST 500.000,APO_FAC 50.0000,AXIS_VEL 100.000,AXIS_ACC 100.000,ORI_TYP #VAR,CIRC_TYP #BASE,JERK_FAC 50.0000,GEAR_JERK 100.000,EXAX_IGN 0}
DECL E6POS XP3217={X 328.0,Y 348.0,Z -17.64,A -180,B 0,C 180,S 2,T 10,E1 0.0,E2 0.0,E3 0.0,E4 0.0,E5 0.0,E6 0.0}
DECL FDAT FP3217={TOOL_NO 1,BASE_NO 0,IPO_FRAME #BASE,POINT2[] " "}
DECL LDAT LCPDAT3217={VEL 2.00000,ACC 100.000,APO_DIST 500.000,APO_FAC 50.0000,AXIS_VEL 100.000,AXIS_ACC 100.000,ORI_TYP #VAR,CIRC_TYP #BASE,JERK_FAC 50.0000,GEAR_JERK 100.000,EXAX_IGN 0}
DECL E6POS XP3218={X 329.0,Y 350.0,Z -17.64,A -180,B 0,C 180,S 2,T 10,E1 0.0,E2 0.0,E3 0.0,E4 0.0,E5 0.0,E6 0.0}
DECL FDAT FP3218={TOOL_NO 1,BASE_NO 0,IPO_FRAME #BASE,POINT2[] " "}
DECL LDAT LCPDAT3218={VEL 2.00000,ACC 100.000,APO_DIST 500.000,APO_FAC 50.0000,AXIS_VEL 100.000,AXIS_ACC 100.000,ORI_TYP #VAR,CIRC_TYP #BASE,JERK_FAC 50.0000,GEAR_JERK 100.000,EXAX_IGN 0}
DECL E6POS XP3219={X 329.0,Y 350.0,Z -17.64,A -180,B 0,C 180,S 2,T 10,E1 0.0,E2 0.0,E3 0.0,E4 0.0,E5 0.0,E6 0.0}
DECL FDAT FP3219={TOOL_NO 1,BASE_NO 0,IPO_FRAME #BASE,POINT2[] " "}
DECL LDAT LCPDAT3219={VEL 2.00000,ACC 100.000,APO_DIST 500.000,APO_FAC 50.0000,AXIS_VEL 100.000,AXIS_ACC 100.000,ORI_TYP #VAR,CIRC_TYP #BASE,JERK_FAC 50.0000,GEAR_JERK 100.000,EXAX_IGN 0}
DECL E6POS XP3220={X 333.0,Y 354.0,Z -17.64,A -180,B 0,C 180,S 2,T 10,E1 0.0,E2 0.0,E3 0.0,E4 0.0,E5 0.0,E6 0.0}
DECL FDAT FP3220={TOOL_NO 1,BASE_NO 0,IPO_FRAME #BASE,POINT2[] " "}
DECL LDAT LCPDAT3220={VEL 2.00000,ACC 100.000,APO_DIST 500.000,APO_FAC 50.0000,AXIS_VEL 100.000,AXIS_ACC 100.000,ORI_TYP #VAR,CIRC_TYP #BASE,JERK_FAC 50.0000,GEAR_JERK 100.000,EXAX_IGN 0}
DECL E6POS XP3221={X 333.0,Y 354.0,Z -17.64,A -180,B 0,C 180,S 2,T 10,E1 0.0,E2 0.0,E3 0.0,E4 0.0,E5 0.0,E6 0.0}
DECL FDAT FP3221={TOOL_NO 1,BASE_NO 0,IPO_FRAME #BASE,POINT2[] " "}
DECL LDAT LCPDAT3221={VEL 2.00000,ACC 100.000,APO_DIST 500.000,APO_FAC 50.0000,AXIS_VEL 100.000,AXIS_ACC 100.000,ORI_TYP #VAR,CIRC_TYP #BASE,JERK_FAC 50.0000,GEAR_JERK 100.000,EXAX_IGN 0}
DECL E6POS XP3222={X 335.0,Y 355.0,Z -17.64,A -180,B 0,C 180,S 2,T 10,E1 0.0,E2 0.0,E3 0.0,E4 0.0,E5 0.0,E6 0.0}
DECL FDAT FP3222={TOOL_NO 1,BASE_NO 0,IPO_FRAME #BASE,POINT2[] " "}
DECL LDAT LCPDAT3222={VEL 2.00000,ACC 100.000,APO_DIST 500.000,APO_FAC 50.0000,AXIS_VEL 100.000,AXIS_ACC 100.000,ORI_TYP #VAR,CIRC_TYP #BASE,JERK_FAC 50.0000,GEAR_JERK 100.000,EXAX_IGN 0}
DECL E6POS XP3223={X 335.0,Y 355.0,Z -17.64,A -180,B 0,C 180,S 2,T 10,E1 0.0,E2 0.0,E3 0.0,E4 0.0,E5 0.0,E6 0.0}
DECL FDAT FP3223={TOOL_NO 1,BASE_NO 0,IPO_FRAME #BASE,POINT2[] " "}
DECL LDAT LCPDAT3223={VEL 2.00000,ACC 100.000,APO_DIST 500.000,APO_FAC 50.0000,AXIS_VEL 100.000,AXIS_ACC 100.000,ORI_TYP #VAR,CIRC_TYP #BASE,JERK_FAC 50.0000,GEAR_JERK 100.000,EXAX_IGN 0}
DECL E6POS XP3224={X 337.0,Y 355.0,Z -17.64,A -180,B 0,C 180,S 2,T 10,E1 0.0,E2 0.0,E3 0.0,E4 0.0,E5 0.0,E6 0.0}
DECL FDAT FP3224={TOOL_NO 1,BASE_NO 0,IPO_FRAME #BASE,POINT2[] " "}
DECL LDAT LCPDAT3224={VEL 2.00000,ACC 100.000,APO_DIST 500.000,APO_FAC 50.0000,AXIS_VEL 100.000,AXIS_ACC 100.000,ORI_TYP #VAR,CIRC_TYP #BASE,JERK_FAC 50.0000,GEAR_JERK 100.000,EXAX_IGN 0}
DECL E6POS XP3225={X 337.0,Y 355.0,Z -17.64,A -180,B 0,C 180,S 2,T 10,E1 0.0,E2 0.0,E3 0.0,E4 0.0,E5 0.0,E6 0.0}
DECL FDAT FP3225={TOOL_NO 1,BASE_NO 0,IPO_FRAME #BASE,POINT2[] " "}
DECL LDAT LCPDAT3225={VEL 2.00000,ACC 100.000,APO_DIST 500.000,APO_FAC 50.0000,AXIS_VEL 100.000,AXIS_ACC 100.000,ORI_TYP #VAR,CIRC_TYP #BASE,JERK_FAC 50.0000,GEAR_JERK 100.000,EXAX_IGN 0}
DECL E6POS XP3226={X 337.0,Y 353.0,Z -17.64,A -180,B 0,C 180,S 2,T 10,E1 0.0,E2 0.0,E3 0.0,E4 0.0,E5 0.0,E6 0.0}
DECL FDAT FP3226={TOOL_NO 1,BASE_NO 0,IPO_FRAME #BASE,POINT2[] " "}
DECL LDAT LCPDAT3226={VEL 2.00000,ACC 100.000,APO_DIST 500.000,APO_FAC 50.0000,AXIS_VEL 100.000,AXIS_ACC 100.000,ORI_TYP #VAR,CIRC_TYP #BASE,JERK_FAC 50.0000,GEAR_JERK 100.000,EXAX_IGN 0}
DECL E6POS XP3227={X 337.0,Y 353.0,Z -17.64,A -180,B 0,C 180,S 2,T 10,E1 0.0,E2 0.0,E3 0.0,E4 0.0,E5 0.0,E6 0.0}
DECL FDAT FP3227={TOOL_NO 1,BASE_NO 0,IPO_FRAME #BASE,POINT2[] " "}
DECL LDAT LCPDAT3227={VEL 2.00000,ACC 100.000,APO_DIST 500.000,APO_FAC 50.0000,AXIS_VEL 100.000,AXIS_ACC 100.000,ORI_TYP #VAR,CIRC_TYP #BASE,JERK_FAC 50.0000,GEAR_JERK 100.000,EXAX_IGN 0}
DECL E6POS XP3228={X 338.0,Y 352.0,Z -17.64,A -180,B 0,C 180,S 2,T 10,E1 0.0,E2 0.0,E3 0.0,E4 0.0,E5 0.0,E6 0.0}
DECL FDAT FP3228={TOOL_NO 1,BASE_NO 0,IPO_FRAME #BASE,POINT2[] " "}
DECL LDAT LCPDAT3228={VEL 2.00000,ACC 100.000,APO_DIST 500.000,APO_FAC 50.0000,AXIS_VEL 100.000,AXIS_ACC 100.000,ORI_TYP #VAR,CIRC_TYP #BASE,JERK_FAC 50.0000,GEAR_JERK 100.000,EXAX_IGN 0}
DECL E6POS XP3229={X 338.0,Y 352.0,Z -17.64,A -180,B 0,C 180,S 2,T 10,E1 0.0,E2 0.0,E3 0.0,E4 0.0,E5 0.0,E6 0.0}
DECL FDAT FP3229={TOOL_NO 1,BASE_NO 0,IPO_FRAME #BASE,POINT2[] " "}
DECL LDAT LCPDAT3229={VEL 2.00000,ACC 100.000,APO_DIST 500.000,APO_FAC 50.0000,AXIS_VEL 100.000,AXIS_ACC 100.000,ORI_TYP #VAR,CIRC_TYP #BASE,JERK_FAC 50.0000,GEAR_JERK 100.000,EXAX_IGN 0}
DECL E6POS XP3230={X 339.0,Y 347.0,Z -17.64,A -180,B 0,C 180,S 2,T 10,E1 0.0,E2 0.0,E3 0.0,E4 0.0,E5 0.0,E6 0.0}
DECL FDAT FP3230={TOOL_NO 1,BASE_NO 0,IPO_FRAME #BASE,POINT2[] " "}
DECL LDAT LCPDAT3230={VEL 2.00000,ACC 100.000,APO_DIST 500.000,APO_FAC 50.0000,AXIS_VEL 100.000,AXIS_ACC 100.000,ORI_TYP #VAR,CIRC_TYP #BASE,JERK_FAC 50.0000,GEAR_JERK 100.000,EXAX_IGN 0}
DECL E6POS XP3231={X 339.0,Y 347.0,Z -17.64,A -180,B 0,C 180,S 2,T 10,E1 0.0,E2 0.0,E3 0.0,E4 0.0,E5 0.0,E6 0.0}
DECL FDAT FP3231={TOOL_NO 1,BASE_NO 0,IPO_FRAME #BASE,POINT2[] " "}
DECL LDAT LCPDAT3231={VEL 2.00000,ACC 100.000,APO_DIST 500.000,APO_FAC 50.0000,AXIS_VEL 100.000,AXIS_ACC 100.000,ORI_TYP #VAR,CIRC_TYP #BASE,JERK_FAC 50.0000,GEAR_JERK 100.000,EXAX_IGN 0}
DECL E6POS XP3232={X 341.0,Y 349.0,Z -17.64,A -180,B 0,C 180,S 2,T 10,E1 0.0,E2 0.0,E3 0.0,E4 0.0,E5 0.0,E6 0.0}
DECL FDAT FP3232={TOOL_NO 1,BASE_NO 0,IPO_FRAME #BASE,POINT2[] " "}
DECL LDAT LCPDAT3232={VEL 2.00000,ACC 100.000,APO_DIST 500.000,APO_FAC 50.0000,AXIS_VEL 100.000,AXIS_ACC 100.000,ORI_TYP #VAR,CIRC_TYP #BASE,JERK_FAC 50.0000,GEAR_JERK 100.000,EXAX_IGN 0}
DECL E6POS XP3233={X 341.0,Y 349.0,Z -17.64,A -180,B 0,C 180,S 2,T 10,E1 0.0,E2 0.0,E3 0.0,E4 0.0,E5 0.0,E6 0.0}
DECL FDAT FP3233={TOOL_NO 1,BASE_NO 0,IPO_FRAME #BASE,POINT2[] " "}
DECL LDAT LCPDAT3233={VEL 2.00000,ACC 100.000,APO_DIST 500.000,APO_FAC 50.0000,AXIS_VEL 100.000,AXIS_ACC 100.000,ORI_TYP #VAR,CIRC_TYP #BASE,JERK_FAC 50.0000,GEAR_JERK 100.000,EXAX_IGN 0}
DECL E6POS XP3234={X 343.0,Y 352.0,Z -17.64,A -180,B 0,C 180,S 2,T 10,E1 0.0,E2 0.0,E3 0.0,E4 0.0,E5 0.0,E6 0.0}
DECL FDAT FP3234={TOOL_NO 1,BASE_NO 0,IPO_FRAME #BASE,POINT2[] " "}
DECL LDAT LCPDAT3234={VEL 2.00000,ACC 100.000,APO_DIST 500.000,APO_FAC 50.0000,AXIS_VEL 100.000,AXIS_ACC 100.000,ORI_TYP #VAR,CIRC_TYP #BASE,JERK_FAC 50.0000,GEAR_JERK 100.000,EXAX_IGN 0}
DECL E6POS XP3235={X 343.0,Y 352.0,Z -17.64,A -180,B 0,C 180,S 2,T 10,E1 0.0,E2 0.0,E3 0.0,E4 0.0,E5 0.0,E6 0.0}
DECL FDAT FP3235={TOOL_NO 1,BASE_NO 0,IPO_FRAME #BASE,POINT2[] " "}
DECL LDAT LCPDAT3235={VEL 2.00000,ACC 100.000,APO_DIST 500.000,APO_FAC 50.0000,AXIS_VEL 100.000,AXIS_ACC 100.000,ORI_TYP #VAR,CIRC_TYP #BASE,JERK_FAC 50.0000,GEAR_JERK 100.000,EXAX_IGN 0}
DECL E6POS XP3236={X 345.0,Y 355.0,Z -17.64,A -180,B 0,C 180,S 2,T 10,E1 0.0,E2 0.0,E3 0.0,E4 0.0,E5 0.0,E6 0.0}
DECL FDAT FP3236={TOOL_NO 1,BASE_NO 0,IPO_FRAME #BASE,POINT2[] " "}
DECL LDAT LCPDAT3236={VEL 2.00000,ACC 100.000,APO_DIST 500.000,APO_FAC 50.0000,AXIS_VEL 100.000,AXIS_ACC 100.000,ORI_TYP #VAR,CIRC_TYP #BASE,JERK_FAC 50.0000,GEAR_JERK 100.000,EXAX_IGN 0}
DECL E6POS XP3237={X 345.0,Y 355.0,Z -17.64,A -180,B 0,C 180,S 2,T 10,E1 0.0,E2 0.0,E3 0.0,E4 0.0,E5 0.0,E6 0.0}
DECL FDAT FP3237={TOOL_NO 1,BASE_NO 0,IPO_FRAME #BASE,POINT2[] " "}
DECL LDAT LCPDAT3237={VEL 2.00000,ACC 100.000,APO_DIST 500.000,APO_FAC 50.0000,AXIS_VEL 100.000,AXIS_ACC 100.000,ORI_TYP #VAR,CIRC_TYP #BASE,JERK_FAC 50.0000,GEAR_JERK 100.000,EXAX_IGN 0}
DECL E6POS XP3238={X 345.0,Y 358.0,Z -17.64,A -180,B 0,C 180,S 2,T 10,E1 0.0,E2 0.0,E3 0.0,E4 0.0,E5 0.0,E6 0.0}
DECL FDAT FP3238={TOOL_NO 1,BASE_NO 0,IPO_FRAME #BASE,POINT2[] " "}
DECL LDAT LCPDAT3238={VEL 2.00000,ACC 100.000,APO_DIST 500.000,APO_FAC 50.0000,AXIS_VEL 100.000,AXIS_ACC 100.000,ORI_TYP #VAR,CIRC_TYP #BASE,JERK_FAC 50.0000,GEAR_JERK 100.000,EXAX_IGN 0}
DECL E6POS XP3239={X 345.0,Y 358.0,Z -17.64,A -180,B 0,C 180,S 2,T 10,E1 0.0,E2 0.0,E3 0.0,E4 0.0,E5 0.0,E6 0.0}
DECL FDAT FP3239={TOOL_NO 1,BASE_NO 0,IPO_FRAME #BASE,POINT2[] " "}
DECL LDAT LCPDAT3239={VEL 2.00000,ACC 100.000,APO_DIST 500.000,APO_FAC 50.0000,AXIS_VEL 100.000,AXIS_ACC 100.000,ORI_TYP #VAR,CIRC_TYP #BASE,JERK_FAC 50.0000,GEAR_JERK 100.000,EXAX_IGN 0}
DECL E6POS XP3240={X 341.0,Y 362.0,Z -17.64,A -180,B 0,C 180,S 2,T 10,E1 0.0,E2 0.0,E3 0.0,E4 0.0,E5 0.0,E6 0.0}
DECL FDAT FP3240={TOOL_NO 1,BASE_NO 0,IPO_FRAME #BASE,POINT2[] " "}
DECL LDAT LCPDAT3240={VEL 2.00000,ACC 100.000,APO_DIST 500.000,APO_FAC 50.0000,AXIS_VEL 100.000,AXIS_ACC 100.000,ORI_TYP #VAR,CIRC_TYP #BASE,JERK_FAC 50.0000,GEAR_JERK 100.000,EXAX_IGN 0}
DECL E6POS XP3241={X 341.0,Y 362.0,Z -17.64,A -180,B 0,C 180,S 2,T 10,E1 0.0,E2 0.0,E3 0.0,E4 0.0,E5 0.0,E6 0.0}
DECL FDAT FP3241={TOOL_NO 1,BASE_NO 0,IPO_FRAME #BASE,POINT2[] " "}
DECL LDAT LCPDAT3241={VEL 2.00000,ACC 100.000,APO_DIST 500.000,APO_FAC 50.0000,AXIS_VEL 100.000,AXIS_ACC 100.000,ORI_TYP #VAR,CIRC_TYP #BASE,JERK_FAC 50.0000,GEAR_JERK 100.000,EXAX_IGN 0}
DECL E6POS XP3242={X 334.0,Y 365.0,Z -17.64,A -180,B 0,C 180,S 2,T 10,E1 0.0,E2 0.0,E3 0.0,E4 0.0,E5 0.0,E6 0.0}
DECL FDAT FP3242={TOOL_NO 1,BASE_NO 0,IPO_FRAME #BASE,POINT2[] " "}
DECL LDAT LCPDAT3242={VEL 2.00000,ACC 100.000,APO_DIST 500.000,APO_FAC 50.0000,AXIS_VEL 100.000,AXIS_ACC 100.000,ORI_TYP #VAR,CIRC_TYP #BASE,JERK_FAC 50.0000,GEAR_JERK 100.000,EXAX_IGN 0}
DECL E6POS XP3243={X 334.0,Y 365.0,Z -17.64,A -180,B 0,C 180,S 2,T 10,E1 0.0,E2 0.0,E3 0.0,E4 0.0,E5 0.0,E6 0.0}
DECL FDAT FP3243={TOOL_NO 1,BASE_NO 0,IPO_FRAME #BASE,POINT2[] " "}
DECL LDAT LCPDAT3243={VEL 2.00000,ACC 100.000,APO_DIST 500.000,APO_FAC 50.0000,AXIS_VEL 100.000,AXIS_ACC 100.000,ORI_TYP #VAR,CIRC_TYP #BASE,JERK_FAC 50.0000,GEAR_JERK 100.000,EXAX_IGN 0}
DECL E6POS XP3244={X 329.0,Y 368.0,Z -17.64,A -180,B 0,C 180,S 2,T 10,E1 0.0,E2 0.0,E3 0.0,E4 0.0,E5 0.0,E6 0.0}
DECL FDAT FP3244={TOOL_NO 1,BASE_NO 0,IPO_FRAME #BASE,POINT2[] " "}
DECL LDAT LCPDAT3244={VEL 2.00000,ACC 100.000,APO_DIST 500.000,APO_FAC 50.0000,AXIS_VEL 100.000,AXIS_ACC 100.000,ORI_TYP #VAR,CIRC_TYP #BASE,JERK_FAC 50.0000,GEAR_JERK 100.000,EXAX_IGN 0}
DECL E6POS XP3245={X 329.0,Y 368.0,Z -17.64,A -180,B 0,C 180,S 2,T 10,E1 0.0,E2 0.0,E3 0.0,E4 0.0,E5 0.0,E6 0.0}
DECL FDAT FP3245={TOOL_NO 1,BASE_NO 0,IPO_FRAME #BASE,POINT2[] " "}
DECL LDAT LCPDAT3245={VEL 2.00000,ACC 100.000,APO_DIST 500.000,APO_FAC 50.0000,AXIS_VEL 100.000,AXIS_ACC 100.000,ORI_TYP #VAR,CIRC_TYP #BASE,JERK_FAC 50.0000,GEAR_JERK 100.000,EXAX_IGN 0}
DECL E6POS XP3246={X 327.0,Y 370.0,Z -17.64,A -180,B 0,C 180,S 2,T 10,E1 0.0,E2 0.0,E3 0.0,E4 0.0,E5 0.0,E6 0.0}
DECL FDAT FP3246={TOOL_NO 1,BASE_NO 0,IPO_FRAME #BASE,POINT2[] " "}
DECL LDAT LCPDAT3246={VEL 2.00000,ACC 100.000,APO_DIST 500.000,APO_FAC 50.0000,AXIS_VEL 100.000,AXIS_ACC 100.000,ORI_TYP #VAR,CIRC_TYP #BASE,JERK_FAC 50.0000,GEAR_JERK 100.000,EXAX_IGN 0}
DECL E6POS XP3247={X 327.0,Y 370.0,Z -17.64,A -180,B 0,C 180,S 2,T 10,E1 0.0,E2 0.0,E3 0.0,E4 0.0,E5 0.0,E6 0.0}
DECL FDAT FP3247={TOOL_NO 1,BASE_NO 0,IPO_FRAME #BASE,POINT2[] " "}
DECL LDAT LCPDAT3247={VEL 2.00000,ACC 100.000,APO_DIST 500.000,APO_FAC 50.0000,AXIS_VEL 100.000,AXIS_ACC 100.000,ORI_TYP #VAR,CIRC_TYP #BASE,JERK_FAC 50.0000,GEAR_JERK 100.000,EXAX_IGN 0}
DECL E6POS XP3248={X 326.0,Y 372.0,Z -17.64,A -180,B 0,C 180,S 2,T 10,E1 0.0,E2 0.0,E3 0.0,E4 0.0,E5 0.0,E6 0.0}
DECL FDAT FP3248={TOOL_NO 1,BASE_NO 0,IPO_FRAME #BASE,POINT2[] " "}
DECL LDAT LCPDAT3248={VEL 2.00000,ACC 100.000,APO_DIST 500.000,APO_FAC 50.0000,AXIS_VEL 100.000,AXIS_ACC 100.000,ORI_TYP #VAR,CIRC_TYP #BASE,JERK_FAC 50.0000,GEAR_JERK 100.000,EXAX_IGN 0}
DECL E6POS XP3249={X 326.0,Y 372.0,Z -17.64,A -180,B 0,C 180,S 2,T 10,E1 0.0,E2 0.0,E3 0.0,E4 0.0,E5 0.0,E6 0.0}
DECL FDAT FP3249={TOOL_NO 1,BASE_NO 0,IPO_FRAME #BASE,POINT2[] " "}
DECL LDAT LCPDAT3249={VEL 2.00000,ACC 100.000,APO_DIST 500.000,APO_FAC 50.0000,AXIS_VEL 100.000,AXIS_ACC 100.000,ORI_TYP #VAR,CIRC_TYP #BASE,JERK_FAC 50.0000,GEAR_JERK 100.000,EXAX_IGN 0}
DECL E6POS XP3250={X 326.0,Y 374.0,Z -17.64,A -180,B 0,C 180,S 2,T 10,E1 0.0,E2 0.0,E3 0.0,E4 0.0,E5 0.0,E6 0.0}
DECL FDAT FP3250={TOOL_NO 1,BASE_NO 0,IPO_FRAME #BASE,POINT2[] " "}
DECL LDAT LCPDAT3250={VEL 2.00000,ACC 100.000,APO_DIST 500.000,APO_FAC 50.0000,AXIS_VEL 100.000,AXIS_ACC 100.000,ORI_TYP #VAR,CIRC_TYP #BASE,JERK_FAC 50.0000,GEAR_JERK 100.000,EXAX_IGN 0}
DECL E6POS XP3251={X 326.0,Y 374.0,Z -17.64,A -180,B 0,C 180,S 2,T 10,E1 0.0,E2 0.0,E3 0.0,E4 0.0,E5 0.0,E6 0.0}
DECL FDAT FP3251={TOOL_NO 1,BASE_NO 0,IPO_FRAME #BASE,POINT2[] " "}
DECL LDAT LCPDAT3251={VEL 2.00000,ACC 100.000,APO_DIST 500.000,APO_FAC 50.0000,AXIS_VEL 100.000,AXIS_ACC 100.000,ORI_TYP #VAR,CIRC_TYP #BASE,JERK_FAC 50.0000,GEAR_JERK 100.000,EXAX_IGN 0}
DECL E6POS XP3252={X 325.0,Y 376.0,Z -17.64,A -180,B 0,C 180,S 2,T 10,E1 0.0,E2 0.0,E3 0.0,E4 0.0,E5 0.0,E6 0.0}
DECL FDAT FP3252={TOOL_NO 1,BASE_NO 0,IPO_FRAME #BASE,POINT2[] " "}
DECL LDAT LCPDAT3252={VEL 2.00000,ACC 100.000,APO_DIST 500.000,APO_FAC 50.0000,AXIS_VEL 100.000,AXIS_ACC 100.000,ORI_TYP #VAR,CIRC_TYP #BASE,JERK_FAC 50.0000,GEAR_JERK 100.000,EXAX_IGN 0}
DECL E6POS XP3253={X 325.0,Y 376.0,Z -17.64,A -180,B 0,C 180,S 2,T 10,E1 0.0,E2 0.0,E3 0.0,E4 0.0,E5 0.0,E6 0.0}
DECL FDAT FP3253={TOOL_NO 1,BASE_NO 0,IPO_FRAME #BASE,POINT2[] " "}
DECL LDAT LCPDAT3253={VEL 2.00000,ACC 100.000,APO_DIST 500.000,APO_FAC 50.0000,AXIS_VEL 100.000,AXIS_ACC 100.000,ORI_TYP #VAR,CIRC_TYP #BASE,JERK_FAC 50.0000,GEAR_JERK 100.000,EXAX_IGN 0}
DECL E6POS XP3254={X 327.0,Y 378.0,Z -17.64,A -180,B 0,C 180,S 2,T 10,E1 0.0,E2 0.0,E3 0.0,E4 0.0,E5 0.0,E6 0.0}
DECL FDAT FP3254={TOOL_NO 1,BASE_NO 0,IPO_FRAME #BASE,POINT2[] " "}
DECL LDAT LCPDAT3254={VEL 2.00000,ACC 100.000,APO_DIST 500.000,APO_FAC 50.0000,AXIS_VEL 100.000,AXIS_ACC 100.000,ORI_TYP #VAR,CIRC_TYP #BASE,JERK_FAC 50.0000,GEAR_JERK 100.000,EXAX_IGN 0}
DECL E6POS XP3255={X 327.0,Y 378.0,Z -17.64,A -180,B 0,C 180,S 2,T 10,E1 0.0,E2 0.0,E3 0.0,E4 0.0,E5 0.0,E6 0.0}
DECL FDAT FP3255={TOOL_NO 1,BASE_NO 0,IPO_FRAME #BASE,POINT2[] " "}
DECL LDAT LCPDAT3255={VEL 2.00000,ACC 100.000,APO_DIST 500.000,APO_FAC 50.0000,AXIS_VEL 100.000,AXIS_ACC 100.000,ORI_TYP #VAR,CIRC_TYP #BASE,JERK_FAC 50.0000,GEAR_JERK 100.000,EXAX_IGN 0}
DECL E6POS XP3256={X 329.0,Y 379.0,Z -17.64,A -180,B 0,C 180,S 2,T 10,E1 0.0,E2 0.0,E3 0.0,E4 0.0,E5 0.0,E6 0.0}
DECL FDAT FP3256={TOOL_NO 1,BASE_NO 0,IPO_FRAME #BASE,POINT2[] " "}
DECL LDAT LCPDAT3256={VEL 2.00000,ACC 100.000,APO_DIST 500.000,APO_FAC 50.0000,AXIS_VEL 100.000,AXIS_ACC 100.000,ORI_TYP #VAR,CIRC_TYP #BASE,JERK_FAC 50.0000,GEAR_JERK 100.000,EXAX_IGN 0}
DECL E6POS XP3257={X 329.0,Y 379.0,Z -17.64,A -180,B 0,C 180,S 2,T 10,E1 0.0,E2 0.0,E3 0.0,E4 0.0,E5 0.0,E6 0.0}
DECL FDAT FP3257={TOOL_NO 1,BASE_NO 0,IPO_FRAME #BASE,POINT2[] " "}
DECL LDAT LCPDAT3257={VEL 2.00000,ACC 100.000,APO_DIST 500.000,APO_FAC 50.0000,AXIS_VEL 100.000,AXIS_ACC 100.000,ORI_TYP #VAR,CIRC_TYP #BASE,JERK_FAC 50.0000,GEAR_JERK 100.000,EXAX_IGN 0}
DECL E6POS XP3258={X 333.0,Y 380.0,Z -17.64,A -180,B 0,C 180,S 2,T 10,E1 0.0,E2 0.0,E3 0.0,E4 0.0,E5 0.0,E6 0.0}
DECL FDAT FP3258={TOOL_NO 1,BASE_NO 0,IPO_FRAME #BASE,POINT2[] " "}
